// Optimizes request count per object.
// > If a single object has more than one request, these multiple requests can be handled via a single RPM-request.
METHOD PRIVATE OptimizeCOV : BOOL
VAR
	i : UDINT;
	j : UDINT;
	bSkipCov : BOOL;
END_VAR
IF (nReqList > 0) THEN
	FOR i:=0 TO nReqList-1 DO
		IF stReqList[i].iReq <> 0 AND_THEN F_IsCovReqType(stReqList[i].iReq) AND_THEN stReqList[i].fbCov^.Master = 0 THEN
			bSkipCov := F_IsCovProperty(stReqList[i].fbCov^.iObject.ObjectType, stReqList[i].fbCov^.ePropID);
			FOR j:=i+1 TO nReqList-1 DO
				IF stReqList[j].iReq <> 0 AND_THEN F_IsCovReqType(stReqList[j].iReq) AND_THEN stReqList[i].fbCov^.iObject.ObjectID = stReqList[j].fbCov^.iObject.ObjectID THEN
					 stReqList[i].fbCov^.AddCovSlave(stReqList[j].fbCov);
					 stReqList[j].fbCov^.Master:=stReqList[i].fbCov;
					 IF stReqList[j].fbCov^.fCOVIncrement = 0 AND F_IsCovProperty(stReqList[j].fbCov^.iObject.ObjectType, stReqList[j].fbCov^.ePropID) THEN
						 IF bSkipCov THEN
						 	stReqList[j].fbCov^.SendSubscription:=FALSE;
						 ELSE
							 bSkipCov:=TRUE;
						 END_IF
					 END_IF
				END_IF
			END_FOR
		END_IF
	END_FOR
END_IF
END_METHOD

// Called after online change.
{attribute 'call_after_online_change_slot' := '10'}
METHOD PROTECTED OnPostOnlineChange
IF iServer <> 0 THEN
	FW_SafeRelease(ADR(iServer));
	iServer:=0;
END_IF
IF iClient <> 0 THEN
	FW_SafeRelease(ADR(iClient));
	iClient:=0;
END_IF
iDevice:=0;

State:=E_BACnetRM_ClientState.eReInit;
END_METHOD

METHOD FB_Exit : BOOL
VAR_INPUT
	 bInCopyCode : BOOL; // if TRUE, the exit method is called for exiting an instance that is copied afterwards (online change).
END_VAR
IF iServer <> 0 THEN
	iServer.OnPlcAction(E_BACnet_PlcAction.eSuspend);
	iServer:=0;
END_IF
IF iClient <> 0 THEN
	FW_SafeRelease(ADR(iClient));
	iClient:=0;
END_IF

iDevice:=0;

DeleteReqList();

IF stReadList <> 0 THEN
	__DELETE(stReadList);
	stReadList:=0;
END_IF
IF stWriteList <> 0 THEN
	__DELETE(stWriteList);
	stWriteList:=0;
END_IF
END_METHOD

PROPERTY Error : BOOL
GET
Error := (eErrorID <> E_BACnet_Error.eNoError);
END_GET
END_PROPERTY

PROPERTY ObjectID : T_BACnet_ObjectIdentifier
GET
ObjectID := tObjectID;
END_GET
END_PROPERTY

PROPERTY ObjectInstance : UDINT
GET
ObjectInstance := nDeviceInstance;
END_GET
END_PROPERTY

PROPERTY ObjectType : E_BACnetObjType
GET
ObjectType := E_BACnetObjType.ObjDevice;
END_GET
END_PROPERTY

PROPERTY OpenRequestCount : UDINT
GET
OpenRequestCount:=nOpenReq;
END_GET
SET
nOpenReq:=OpenRequestCount;
END_SET
END_PROPERTY

PROPERTY ReadMode : E_BACnet_CommMode
GET
ReadMode:=eReadMode;
END_GET
SET
eReadMode:=ReadMode;
END_SET
END_PROPERTY

PROPERTY Ready : BOOL
GET
Ready := bReady;
END_GET
END_PROPERTY

PROPERTY State : E_BACnetRM_ClientState
GET
State := eState;
END_GET
SET
PRIVATE 
VAR
END_VAR
IF (State = E_BACnetRM_ClientState.eError) THEN
	_tReInitTime := TIME();
END_IF

eState := State;
END_SET
END_PROPERTY

END_FUNCTION_BLOCK

// POUs/Remote/Requests/[Internal]/FB_BACnetRM_ReqFifo
{attribute 'c++_compatible'}
{attribute 'enable_dynamic_creation'}
{attribute 'hide'}
FUNCTION_BLOCK FB_BACnetRM_ReqFifo EXTENDS FB_BACnetRM_ReqBase
VAR_INPUT
	bRpm : BOOL;
	bWpm : BOOL;
END_VAR
VAR
	pReqFifo	: POINTER TO ST_BACnetRM_FifoEntry;
	nReqFifo	: UDINT := 0;
	nMaxFifo	: UDINT := 0;
	nPendFifo	: UDINT := 0;
END_VAR

METHOD INTERNAL AddFifoReq : BOOL
VAR_INPUT
	pEntry : ST_BACnetRM_FifoEntry;
END_VAR
VAR
	nTmp : UDINT;
	nTmpSize : UDINT;
	pTmp : POINTER TO ST_BACnetRM_FifoEntry;
END_VAR
IF nReqFifo+1 >= nMaxFifo THEN
	nTmp := 2*nMaxFifo+100;
	nTmpSize := nTmp*SIZEOF(ST_BACnetRM_FifoEntry);
	pTmp := __NEW(BYTE,nTmpSize);
	IF pTmp = 0 THEN
		RETURN;
	END_IF
	IF pReqFifo <> 0 THEN
		MEMCPY(pTmp, pReqFifo, nMaxFifo*SIZEOF(ST_BACnetRM_FifoEntry));
		__DELETE(pReqFifo);
	END_IF
	pReqFifo:=pTmp;
	nMaxFifo:=nTmp;
END_IF

pReqFifo[nReqFifo]:=pEntry;
nReqFifo:=nReqFifo+1;

AddFifoReq:=TRUE;
END_METHOD

METHOD INTERNAL ProcessReadFifo : BOOL
VAR_INPUT
END_VAR
VAR
	pRequest : ST_BACnetRM_ReqPtr;
	nSize : UDINT;
	n :UDINT;
	pEntries : POINTER TO ST_BACnetRM_ReadEntry;	
	x : UDINT;
	iTmpFB : I_BACnetRM_BasicReq;
END_VAR
IF Valid THEN
	WHILE Client.nOpenReq < Client.nMaxParallelRequests AND nReqFifo > 0 DO		
		IF bRpm AND nReqFifo>1 THEN
			n:=0;
			nSize:=MIN(nReqFifo, Client.nRPMPropertiesPerRequest)*SIZEOF(ST_BACnetRM_ReadEntry);
			pRequest.fbRpm := __NEW(FB_BACnetRM_ReqRpm);
			IF pRequest.fbRpm = 0 THEN
				RETURN;
			END_IF
			pEntries:=__NEW(BYTE,nSize);
			IF pEntries = 0 THEN
				__DELETE(pRequest.fbRpm);
				RETURN;
			END_IF
			WHILE n<nReqFifo AND n < Client.nRPMPropertiesPerRequest DO
				pEntries[n].iObject:=pReqFifo[n].fbRead^.iObject;
				pEntries[n].ePropID:=pReqFifo[n].fbRead^.ePropID;
				pEntries[n].pData:=pReqFifo[n].fbRead^.pData;
				pEntries[n].nData:=pReqFifo[n].fbRead^.nData;
				pEntries[n].nIndex:=pReqFifo[n].fbRead^.nIndex;
				IF __QUERYINTERFACE(pReqFifo[0].fbRead^, iTmpFB) THEN
					pEntries[n].iReadFB:=iTmpFB;
				END_IF
				n:=n+1;
			END_WHILE		
			pRequest.fbRpm^(Client:=Client, iObject:=pReqFifo[0].fbRead^.iObject, pEntries:=pEntries, nEntries:=n, bFreeEntries:=TRUE);
			IF pRequest.fbRpm^.UpdateRequest() AND_THEN pRequest.fbRpm^.Send() THEN
				Client.OpenRequestCount:=Client.nOpenReq+1;
				pReqFifo[0].fbRead^.Request:=pRequest;
				pReqFifo[0].fbRead^.bRequestRPM:=TRUE;
				IF nReqFifo-n > 0 THEN
					MEMMOVE(pReqFifo, ADR(pReqFifo[n]), (nReqFifo-n)*SIZEOF(ST_BACnetRM_ReadEntry));
				END_IF
				nReqFifo:=nReqFifo-n;
			ELSE
				__DELETE(pRequest.fbRpm);
				RETURN;
			END_IF
		ELSE
			pRequest.fbRead := __NEW(FB_BACnetRM_ReqRead);
			IF pRequest.fbRead = 0 THEN
				RETURN;
			END_IF
			__QUERYINTERFACE(pReqFifo[0].fbRead^, iTmpFB);
			pRequest.fbRead^(Client:=Client, iObject:=pReqFifo[0].fbRead^.iObject, pData:=pReqFifo[0].fbRead^.pData, nData:=pReqFifo[0].fbRead^.nData, ePropID:=pReqFifo[0].fbRead^.ePropID, iReadFB:=iTmpFB);
			Client.OpenRequestCount:=Client.nOpenReq+1;
			pReqFifo[0].fbRead^.Request:=pRequest;	
			pReqFifo[0].fbRead^.bRequestRPM:=FALSE;
			IF pRequest.fbRead^.Send() THEN
				IF nReqFifo-n > 0 THEN
					MEMMOVE(pReqFifo, ADR(pReqFifo[1]),(nReqFifo-1)*SIZEOF(ST_BACnetRM_ReadEntry));
				END_IF
				nReqFifo:=nReqFifo-1;
			ELSE
				Client.OpenRequestCount:=Client.nOpenReq-1;
				__DELETE(pRequest.fbRead);
				RETURN;
			END_IF
		END_IF
	END_WHILE
	
	ProcessReadFifo:=TRUE;
ELSE
	// (BETA) ... Output Error
END_IF
END_METHOD

METHOD INTERNAL ProcessWriteFifo : BOOL
VAR_INPUT
END_VAR
VAR
	pRequest : ST_BACnetRM_ReqPtr;
	nSize : UDINT;
	n : UDINT;
	pEntries : POINTER TO ST_BACnetRM_WriteEntry;
	iTmpFB : I_BACnetRM_BasicReq;
END_VAR
IF Valid THEN
	WHILE Client.nOpenReq < Client.nMaxParallelRequests AND nReqFifo > 0 DO		
		IF bWpm THEN
			n:=0;
			nSize:=MIN(nReqFifo, Client.nRPMPropertiesPerRequest)*SIZEOF(ST_BACnetRM_WriteEntry);
			pRequest.fbWpm:= __NEW(FB_BACnetRM_ReqWpm);
			IF pRequest.fbWpm = 0 THEN
				RETURN;
			END_IF
			pEntries:=__NEW(BYTE,nSize);
			IF pEntries = 0 THEN
				__DELETE(pRequest.fbWpm);
				RETURN;
			END_IF
			WHILE n<nReqFifo-1 AND n < Client.nRPMPropertiesPerRequest DO
				pEntries[n].iObject:=pReqFifo[n].fbWrite^.iObject;
				pEntries[n].ePropID:=pReqFifo[n].fbWrite^.ePropID;
				pEntries[n].pData:=pReqFifo[n].fbWrite^.pData;
				pEntries[n].nData:=pReqFifo[n].fbWrite^.nData;
				pEntries[n].nIndex:=pReqFifo[n].fbWrite^.nIndex;
				IF __QUERYINTERFACE(pReqFifo[0].fbWrite^, iTmpFB) THEN
					pEntries[n].iWriteFB:=iTmpFB;
				END_IF
				n:=n+1;
			END_WHILE
			pRequest.fbWpm^(Client:=Client, pEntries:=pEntries, nEntries:=n, bFreeEntries:=TRUE);
			IF pRequest.fbWpm^.UpdateRequest() AND_THEN pRequest.fbWpm^.Send() THEN
				Client.OpenRequestCount:=Client.nOpenReq+1;
				pReqFifo[0].fbRead^.Request:=pRequest;
				pReqFifo[0].fbWrite^.bRequestWPM:=TRUE;
				IF nReqFifo-n > 0 THEN
					MEMMOVE(pReqFifo, ADR(pReqFifo[n]), (nReqFifo-n)*SIZEOF(ST_BACnetRM_WriteEntry));
				END_IF
				nReqFifo:=nReqFifo-n;
			ELSE
				__DELETE(pRequest.fbWpm);
				RETURN;
			END_IF
		ELSE
			pRequest.fbWrite := __NEW(FB_BACnetRM_ReqWrite);
			IF pRequest.fbWrite = 0 THEN
				RETURN;
			END_IF
			pRequest.fbWrite^.pData:=pReqFifo[0].fbWrite^.pData;
			pRequest.fbWrite^.nData:=pReqFifo[0].fbWrite^.nData;
			__QUERYINTERFACE(pReqFifo[0].fbWrite^, iTmpFB);
			pRequest.fbWrite^(Client:=Client, iObject:=pReqFifo[0].fbWrite^.iObject, ePropID:=pReqFifo[0].fbWrite^.ePropID, iWriteFB:=iTmpFB);
			IF pRequest.fbWrite^.Send() THEN
				pReqFifo[0].fbWrite^.Request:=pRequest;	
				pReqFifo[0].fbWrite^.bRequestWPM:=FALSE;
				Client.OpenRequestCount:=Client.nOpenReq+1;
				IF (nReqFifo-1) > 0 THEN
					MEMMOVE(pReqFifo, ADR(pReqFifo[1]),(nReqFifo-1)*SIZEOF(ST_BACnetRM_WriteEntry));
				END_IF
				nReqFifo:=nReqFifo-1;
			ELSE
				__DELETE(pRequest.fbWrite);
				RETURN;
			END_IF
		END_IF
	END_WHILE
	
	ProcessWriteFifo:=TRUE;
ELSE
	// (BETA) ... Output Error
END_IF
END_METHOD

METHOD FB_Exit : BOOL
VAR_INPUT
	 bInCopyCode : BOOL; // if TRUE, the exit method is called for exiting an instance that is copied afterwards (online change).
END_VAR
IF pReqFifo <> 0 THEN
	__DELETE(pReqFifo);
	pReqFifo:=0;
END_IF
END_METHOD

PROPERTY Valid : BOOL
GET
// Hint:
// > Don't call "super()"!
//   The "iObject" Interface-pointer is ignored to this instance because it is unused.
Valid := (__ISVALIDREF(Client));
END_GET
END_PROPERTY

END_FUNCTION_BLOCK

// POUs/Remote/Requests/[Internal]/[Base]/FB_BACnetRM_ReqBase
{attribute 'c++_compatible'}
{attribute 'enable_dynamic_creation'}
{attribute 'hide'}
FUNCTION_BLOCK FB_BACnetRM_ReqBase IMPLEMENTS I_BACnetRM_BaseReq
VAR_INPUT
	{attribute 'initialize_on_call'}
	{attribute 'no_copy'}
	Client : REFERENCE TO FB_BACnet_Client;
	iObject : I_BACnetRM_BaseObject;
END_VAR

METHOD PROTECTED OnError
VAR_INPUT
	stResult		: POINTER TO SendDataRequestResult;
	sLogCode		: STRING			:= '';
END_VAR
VAR
	i : UDINT;
END_VAR
IF (iObject <> 0) THEN
	iObject.OnReqError(THIS^, stResult, 'OE01');
END_IF
END_METHOD

METHOD GetRequestType : E_BACnetRM_RequestType
VAR_INPUT
END_VAR
GetRequestType:=E_BACnetRM_RequestType.eUndefined;
END_METHOD

METHOD IsReady : BOOL
END_METHOD

PROPERTY Valid : BOOL
GET
VAR
	iTest : BOOL;
END_VAR
Valid := (__ISVALIDREF(Client)) AND (iObject <> 0);
END_GET
END_PROPERTY

METHOD Send : BOOL
VAR
	_ClTmp : ITcIoBACnetPlcClient;
END_VAR
END_METHOD

END_FUNCTION_BLOCK

// POUs/Remote/Requests/[Internal]/FB_BACnetRM_ReqRpm
{attribute 'c++_compatible'}
{attribute 'enable_dynamic_creation'}
{attribute 'hide'}
FUNCTION_BLOCK FB_BACnetRM_ReqRpm EXTENDS FB_BACnetRM_ReqBasic
VAR_INPUT
	pEntries : POINTER TO ST_BACnetRM_ReadEntry;
	nEntries : UDINT;
	bFreeEntries : BOOL; 
END_VAR
VAR_OUTPUT
	bInit : BOOL;
END_VAR
VAR 
	req : SendDataRequest;
	pTmp : POINTER TO ST_BACnetRM_RpmListEntry;
END_VAR

IF NOT __ISVALIDREF(Client) THEN
	bError:=TRUE;
END_IF

SUPER^();

{attribute 'hide'}
METHOD Send : BOOL
IF Valid THEN
	IF stReq = 0 THEN
		RETURN;
	END_IF
	
	Send:=SUPER^.Send();
END_IF
END_METHOD

METHOD INTERNAL UpdateRequest : BOOL
VAR_INPUT
END_VAR
VAR
	nSize : UDINT;
	i : UDINT;
	nTmpSize : UDINT;
END_VAR
IF Valid THEN
	IF stReq <> 0 AND_THEN stReq^.pData <> 0 THEN
		pTmp:=stReq^.pData;
		__DELETE(pTmp);
		stReq^.pData:=0;
	END_IF
	nTmpSize := SIZEOF(ST_BACnetRM_RpmListEntry)*nEntries;
	pTmp := __NEW(BYTE,nTmpSize);
	IF pTmp = 0 THEN
		RETURN;
	END_IF
	
	FOR i:=0 TO nEntries-1 DO
		pTmp[i].tObjectID := pEntries[i].iObject.ObjectID;
		pTmp[i].ePropID := pEntries[i].ePropID;
		pTmp[i].nArrayIndex := 0;
		pTmp[i].nValidBits := 0;
		pTmp[i].nPriority := 0;
		pTmp[i].nEntrySize := SIZEOF(ST_BACnetRM_RpmListEntry) - 8;
		IF i <> nEntries -1 THEN
			pTmp[i].nEntrySize := pTmp[i].nEntrySize + 16#80000000;
		END_IF
	END_FOR
	
	stReq := ADR(req);
	stReq^.pData := pTmp;
	stReq^.nData := nTmpSize;
	
	stReq^.service := E_BACnetConfirmedService.SrvReadPropertyMultiple;
	stReq^.deviceId := Client.ObjectInstance;
	
	bInit:=TRUE;
	
	UpdateRequest:=TRUE;
ELSE
	// (BETA) ... Output Error
END_IF
END_METHOD

METHOD PRIVATE Free
VAR_INPUT
END_VAR
IF bFreeEntries AND pEntries <> 0 THEN
	__DELETE(pEntries);
	pEntries:=0;
	bFreeEntries:=FALSE;
END_IF

IF stReq <> 0 AND_THEN stReq^.pData <> 0 THEN
	pTmp:=req.pData;
	__DELETE(pTmp);
	req.pData:=0;
	stReq:=0;
END_IF
END_METHOD

METHOD PROTECTED OnError
VAR_INPUT
	stResult		: POINTER TO SendDataRequestResult;
	sLogCode		: STRING			:= '';
END_VAR
VAR
	i : UDINT;
END_VAR
// Do not call super! Handle each entry's error:
// SUPER^.OnError(eResult, sLogCode);

FOR i:=0 TO nEntries-1 DO
	IF pEntries[i].iReadFB <> 0 THEN
		pEntries[i].iReadFB.SetError();
		IF (pEntries[i].iObject <> 0) THEN
			pEntries[i].iObject.OnReqError(THIS^, stResult, 'OE07');
		END_IF	
	END_IF
END_FOR
END_METHOD

METHOD PROTECTED ProcessResult : HRESULT
VAR_INPUT
	pResult	: POINTER TO SendDataRequestResult;
END_VAR
VAR
	pPropList : POINTER TO ST_BACnetRM_RpmListEntry;
	i : UDINT;
END_VAR
IF pResult^.service <> E_BACnetConfirmedService.SrvReadPropertyMultiple THEN
	ProcessResult:=E_FAIL;
	RETURN;
END_IF

IF pEntries = 0 THEN // Request object has already been deleted
	ProcessResult:=E_FAIL;
	RETURN;
END_IF

// set all entries to error, all good entries in response will be set to good afterwards
FOR i:=0 TO nEntries-1 DO
	IF pEntries[i].iReadFB <> 0 THEN
		pEntries[i].iReadFB.SetError();
	END_IF
	
	pEntries[i]._bError := TRUE;
END_FOR

// copy data:
pPropList := pResult^.pData;
WHILE pPropList <> 0 DO
	_WritePropEntry(pPropList);
	pPropList := F_BACnet_NextListElem(pPropList, pPropList^.nEntrySize);
END_WHILE

// Evaluate remaining errors:
FOR i:=0 TO nEntries-1 DO
	IF (pEntries[i]._bError) AND_THEN (pEntries[i].iObject <> 0) THEN
		pEntries[i].iObject.OnReqError(THIS^, pResult, 'OE28');
	END_IF
END_FOR

ProcessResult:=S_OK;
END_METHOD

METHOD PRIVATE _WritePropEntry : BOOL
VAR_INPUT
	pEntry : POINTER TO ST_BACnetRM_RpmListEntry;
END_VAR
VAR
	i : UDINT;
END_VAR
FOR i:=0 TO nEntries-1 DO
	IF (pEntries[i].iObject.ObjectID = pEntry^.tObjectID) AND (pEntries[i].ePropID = pEntry^.ePropID) THEN
		CopyRemoteData(pEntries[i].iObject, pEntry^.ePropID ,pEntries[i].pData, pEntries[i].nData, F_BACnet_EndOf(pEntry, SIZEOF(ST_BACnetRM_RpmListEntry)), F_BACnet_ElemSize(pEntry^.nEntrySize)-16); 
		IF pEntries[i].iReadFB <> 0 THEN
			pEntries[i].iReadFB.SetReady();
		END_IF
		pEntries[i]._bError := FALSE;
		
		_WritePropEntry:=TRUE;
	END_IF
END_FOR
END_METHOD

METHOD FB_exit : BOOL
VAR_INPUT
	bInCopyCode : BOOL; // if TRUE, the exit method is called for exiting an instance that is copied afterwards (online change).
END_VAR
Free();
END_METHOD

METHOD GetRequestType : E_BACnetRM_RequestType
VAR_INPUT
END_VAR
GetRequestType := E_BACnetRM_RequestType.eReadPropertyMultiple;
END_METHOD

END_FUNCTION_BLOCK

// POUs/Remote/Requests/[Internal]/[Base]/FB_BACnetRM_ReqBasic
{attribute 'c++_compatible'}
{attribute 'enable_dynamic_creation'}
{attribute 'hide'}
FUNCTION_BLOCK FB_BACnetRM_ReqBasic EXTENDS FB_BACnetRM_ReqBase IMPLEMENTS ITcIoBACnetServiceResponseSink
VAR_INPUT
	tCycleTime : TIME := T#5S;
END_VAR
VAR_OUTPUT
	bBusy : BOOL;
	bError : BOOL;
	bReady : BOOL;
END_VAR
VAR
	{attribute 'hide'}
	stReq : POINTER TO SendDataRequest;
	timer : TON;
END_VAR

{attribute 'c++_compatible'}
{attribute 'minimal_input_size' := '4'}
{attribute 'pack_mode' := '4'}
{attribute 'hide'}
METHOD OnSendPropertyDataRequest : HRESULT
VAR_INPUT
	pResult	: POINTER TO SendDataRequestResult;
END_VAR
IF (Valid) AND_THEN (pResult <> 0) THEN
	IF F_BACnetRM_IsErrorSet(pResult) THEN
		SetError();
		OnError(pResult, 'OSPDR04');
		OnSendPropertyDataRequest:=S_FALSE;
	ELSE
		IF S_OK = ProcessResult(pResult) THEN
			SetReady();
			OnSendPropertyDataRequest:=S_OK;
		ELSE
			OnSendPropertyDataRequest:=S_FALSE;
		END_IF	
	END_IF
	Client.OnRequestComplete();
END_IF
END_METHOD

METHOD INTERNAL InitTimer : BOOL
VAR_INPUT
END_VAR
timer(IN:=FALSE, PT:=T#1MS);
timer(IN:=TRUE, PT:=T#1MS);
END_METHOD

{attribute 'hide'}
METHOD SetBusy
bBusy := TRUE;
bError := FALSE;
bReady := FALSE;
END_METHOD

{attribute 'hide'}
METHOD SetError
bBusy := FALSE;
bError := TRUE;
bReady := FALSE;
END_METHOD

{attribute 'hide'}
METHOD SetReady
bBusy := FALSE;
bError := FALSE;
bReady := TRUE;
END_METHOD

{attribute 'c++_compatible'}
{attribute 'minimal_input_size' := '4'}
{attribute 'pack_mode' := '4'}
{attribute 'hide'}
METHOD TcAddRef : UDINT
END_METHOD

{attribute 'c++_compatible'}
{attribute 'minimal_input_size' := '4'}
{attribute 'pack_mode' := '4'}
{attribute 'hide'}
METHOD TcQueryInterface : HRESULT
VAR_INPUT
	iid	: REFERENCE TO IID;
	pipItf	: POINTER TO PVOID;
END_VAR
VAR
	ipSink : ITcIoBACnetServiceResponseSink;
	ipUnknown : ITcUnknown;	
END_VAR
IF GuidsEqual(ADR(iid), ADR(TC_GLOBAL_IID_LIST.IID_ITcIoBACnetServiceResponseSink)) THEN
	ipSink := THIS^; // cast to interface pointer
	pipItf^ := ITCUNKNOWN_TO_PVOID(ipSink);
	TcAddRef();
	TcQueryInterface := S_OK;
ELSIF GuidsEqual(ADR(iid), ADR(TC_GLOBAL_IID_LIST.IID_ITcUnknown)) THEN
	ipUnknown := THIS^; // cast to interface pointer
	pipItf^ := ITCUNKNOWN_TO_PVOID(ipUnknown);
	TcAddRef();
	TcQueryInterface := S_OK;
ELSE
	TcQueryInterface := E_HRESULTAdsErr.NOINTERFACE ; //Call super if this fb extends some other
END_IF
END_METHOD

{attribute 'c++_compatible'}
{attribute 'minimal_input_size' := '4'}
{attribute 'pack_mode' := '4'}
{attribute 'hide'}
METHOD TcRelease : UDINT
END_METHOD

METHOD PROTECTED CopyRemoteData : BOOL
VAR_INPUT
	iObject : I_BACnetRM_BaseObject;
	ePropID : E_BACnetPropIdentifier;
	pDst : PVOID;
	nDst : UDINT;
	pRead : PVOID;
	nRead : UDINT;
END_VAR
VAR
	i 	 : INT;
	pByte : POINTER TO BYTE;
	pSchedPv : POINTER TO ST_BACnet_ValueList;
END_VAR
// Individual treatment:
CASE (ePropID) OF
	E_BACnetPropIdentifier.PropPresentValue:
		IF iObject.ObjectType = E_BACnetObjType.ObjSchedule THEN
			IF (nRead >= 16) THEN
				pSchedPv := pRead;
				CASE pSchedPv^.listEntry.eValueChoice OF
					E_BACnet_ValueChoice.eBoolValue:
						MEMCPY(pDst, ADR(pSchedPv^.listEntry.stValue), MIN(SIZEOF(BOOL),nDst)); 
					E_BACnet_ValueChoice.eRealValue:
						MEMCPY(pDst, ADR(pSchedPv^.listEntry.stValue), MIN(SIZEOF(REAL),nDst)); 
					E_BACnet_ValueChoice.eUnsignedValue:
						MEMCPY(pDst, ADR(pSchedPv^.listEntry.stValue), MIN(SIZEOF(UDINT),nDst)); 
					E_BACnet_ValueChoice.eEnumerationValue:
						MEMCPY(pDst, ADR(pSchedPv^.listEntry.stValue.enumValue), MIN(SIZEOF(UDINT),nDst)); 
				END_CASE
			
				CopyRemoteData := TRUE;
			END_IF
		END_IF
		
	// Consider enumerations with smaller base-types:
	E_BACnetPropIdentifier.PropCurrentlyActivePriority:
		nRead := nDst;
		
END_CASE

// Check if received bytes match expected size:
IF (NOT CopyRemoteData) AND_THEN (nRead <= nDst) THEN
	// Individual treatment:
	CASE (ePropID) OF
		E_BACnetPropIdentifier.PropStatusFlags:
			pByte:=pDst;
			FOR i:=0 TO 3 DO
				IF F_BACnet_IsBitFieldBitSetPtr(pRead, i) THEN
					pByte[i]:=1;
				ELSE
					pByte[i]:=0;
				END_IF
			END_FOR
			
		E_BACnetPropIdentifier.PropAckedTransitions,
		E_BACnetPropIdentifier.PropEventEnable:
			pByte:=pDst;
			FOR i:=0 TO 2 DO
				IF F_BACnet_IsBitFieldBitSetPtr(pRead, i) THEN
					pByte[i]:=1;
				ELSE
					pByte[i]:=0;
				END_IF
			END_FOR
			
	ELSE
		// Default treatment:
		MEMCPY(pDst, pRead, MIN(nRead,nDst)); 
	END_CASE
	
	CopyRemoteData := TRUE;
END_IF

IF (CopyRemoteData) THEN
	// Notify object about changed value:
	iObject.OnCOV(ePropID);
ELSE
	F_BA_LogMessage3(ADSLOG_MSGTYPE_ERROR, 'CRD51', 'Unable to process remote data due to invalid size (Property: "%d", Read: %d Bytes, Expected: %d Bytes)!', F_INT(ePropID), F_UDINT(nRead), F_UDINT(nDst));
END_IF
END_METHOD

METHOD PROTECTED ProcessResult : HRESULT
VAR_INPUT
	pResult	: POINTER TO SendDataRequestResult;
END_VAR
ProcessResult:=S_OK;
END_METHOD

METHOD Send : BOOL
VAR
	_ClTmp : ITcIoBACnetPlcClient;
END_VAR
IF Valid THEN
	_ClTmp := Client.iClient;
	
	SetBusy();
	IF S_OK = _ClTmp.SendPropertyDataRequest(stReq, THIS^) THEN
		Send:=TRUE;
		StartTimer();
	ELSE
		SetError();
		Send:=FALSE; 
	END_IF
END_IF
END_METHOD

METHOD PROTECTED StartTimer : BOOL
VAR_INPUT
END_VAR
timer(IN:=FALSE, PT:=tCycleTime);
timer(IN:=TRUE, PT:=tCycleTime);
END_METHOD

METHOD GetRequestType : E_BACnetRM_RequestType
VAR_INPUT
END_VAR
GetRequestType:=E_BACnetRM_RequestType.eUndefined;
END_METHOD

METHOD IsReady : BOOL
VAR_INPUT
END_VAR
timer(Q=>IsReady);
IF bBusy THEN
	IsReady:=FALSE;
END_IF
END_METHOD

END_FUNCTION_BLOCK

// POUs/Remote/Requests/[Internal]/FB_BACnetRM_ReqRead
{attribute 'c++_compatible'}
{attribute 'enable_dynamic_creation'}
{attribute 'hide'}
FUNCTION_BLOCK FB_BACnetRM_ReqRead EXTENDS FB_BACnetRM_ReqBasic
VAR_INPUT
	ePropID : E_BACnetPropIdentifier;
	pData : PVOID;
	nData : UDINT;
	iReadFB : I_BACnetRM_BasicReq;
END_VAR
VAR 
	req : SendDataRequest;
END_VAR

IF NOT __ISVALIDREF(Client) THEN
	bError:=TRUE;
END_IF

SUPER^();

{attribute 'hide'}
METHOD Send : BOOL
IF Valid THEN
	IF stReq = 0 THEN
		IF ePropID = E_BACnetPropIdentifier.PropLogBuffer THEN
			req.service := E_BACnetConfirmedService.SrvReadRange;
		ELSE
			req.service := E_BACnetConfirmedService.SrvReadProperty;
		END_IF	
		req.objectIdentifier := iObject.ObjectID;
		req.propertyIdentifier := ePropID;
		req.pData := pData;
		req.nData := nData;
		req.deviceId := Client.ObjectInstance;
		stReq := ADR(req);
	END_IF
	
	Send:=SUPER^.Send();
END_IF
END_METHOD

METHOD PROTECTED OnError
VAR_INPUT
	stResult		: POINTER TO SendDataRequestResult;
	sLogCode		: STRING			:= '';
END_VAR
SUPER^.OnError(stResult, sLogCode);

IF iReadFB <> 0 THEN
	iReadFB.SetError();
END_IF
END_METHOD

METHOD PROTECTED ProcessResult : HRESULT
VAR_INPUT
	pResult	: POINTER TO SendDataRequestResult;
END_VAR
IF Valid THEN
	IF (CopyRemoteData(iObject, ePropID, pData, nData, pResult^.pData, pResult^.nData)) THEN
		IF iReadFB <> 0 THEN
			iReadFB.SetReady();
		END_IF
		ProcessResult:=S_OK;
	ELSE
		IF iReadFB <> 0 THEN
			iReadFB.SetError();
		END_IF
		ProcessResult:=E_FAIL;
	END_IF
END_IF
END_METHOD

METHOD GetRequestType : E_BACnetRM_RequestType
VAR_INPUT
END_VAR
GetRequestType:=E_BACnetRM_RequestType.eRead;
END_METHOD

END_FUNCTION_BLOCK

// POUs/Remote/Requests/[Internal]/FB_BACnetRM_ReqWpm
{attribute 'c++_compatible'}
{attribute 'enable_dynamic_creation'}
{attribute 'hide'}
FUNCTION_BLOCK FB_BACnetRM_ReqWpm EXTENDS FB_BACnetRM_ReqBasic
VAR_INPUT
	pEntries : POINTER TO ST_BACnetRM_WriteEntry;
	nEntries : UDINT;
	bFreeEntries : BOOL; 
END_VAR
VAR_OUTPUT
	bInit : BOOL;
END_VAR
VAR 
	{attribute 'hide'}
	req : SendDataRequest;
	{attribute 'hide'}
	pTmp : POINTER TO ST_BACnetRM_RpmListEntry;
END_VAR

IF NOT __ISVALIDREF(Client) THEN
	bError:=TRUE;
END_IF

SUPER^();

{attribute 'hide'}
METHOD Send : BOOL
IF Valid THEN
	IF stReq = 0 THEN
		Send:=FALSE;
		RETURN;
	END_IF
	
	UpdateRequest();
	Send:=SUPER^.Send();
END_IF
END_METHOD

METHOD INTERNAL UpdateRequest : BOOL
VAR_INPUT
END_VAR
VAR
	nSize : UDINT;
	i : UDINT;
	nTmpSize : UDINT;
	nTmpEntrySize : UDINT;
END_VAR
IF Valid THEN
	IF stReq <> 0 AND_THEN stReq^.pData <> 0 THEN
		pTmp:=stReq^.pData;
		__DELETE(pTmp);
	END_IF
	FOR i:=0 TO nEntries-1 DO
		IF pEntries[i].pEnable = 0 OR_ELSE pEntries[i].pEnable^ > 0 THEN
			nTmpSize := nTmpSize + SIZEOF(ST_BACnetRM_RpmListEntry) + F_BACnet_AlignedSize(F_BACnetRM_GetWriteEntrySize(pEntries[i]));
		END_IF
	END_FOR
	pTmp := __NEW(BYTE,nTmpSize);
	IF pTmp = 0 THEN
		UpdateRequest:=FALSE;
		RETURN;
	END_IF
	
	stReq := ADR(req);
	stReq^.pData := pTmp;
	FOR i:=0 TO nEntries-1 DO
		IF pEntries[i].pEnable = 0 OR_ELSE pEntries[i].pEnable^ > 0 THEN
			pTmp^.tObjectID := pEntries[i].iObject.ObjectID;
			pTmp^.ePropID := pEntries[i].ePropID;
			pTmp^.nArrayIndex := 0;
			pTmp^.nValidBits := 0; 
			IF pEntries[i].nPriority <> 16 THEN
				pTmp^.nValidBits.1 := 1;
				pTmp^.nPriority := pEntries[i].nPriority;
			ELSE
				pTmp^.nPriority := 0;
			END_IF
			nTmpEntrySize := F_BACnetRM_GetWriteEntrySize(pEntries[i]);
			pTmp^.nEntrySize := F_BACnet_AlignedSize(nTmpEntrySize) + SIZEOF(ST_BACnetRM_RpmListEntry) - 8;
			
			IF nTmpEntrySize <> 0 THEN
				MEMCPY(F_BACnet_EndOf(pTmp, SIZEOF(ST_BACnetRM_RpmListEntry)), pEntries[i].pData, pEntries[i].nData); 
			END_IF

			IF i <> nEntries -1 THEN
				pTmp[i].nEntrySize := pTmp[i].nEntrySize + 16#80000000;
			END_IF
			pTmp := F_BACnet_NextListElem(pTmp, pTmp^.nEntrySize);
		END_IF
	END_FOR
	
	stReq^.nData := nTmpSize;
	stReq^.service := E_BACnetConfirmedService.SrvWritePropertyMultiple;
	stReq^.deviceId := Client.ObjectInstance;
	
	bInit:=TRUE;
	
	UpdateRequest:=TRUE;
ELSE
	F_BA_LogMessage(ADSLOG_MSGTYPE_ERROR, 'WPM82', 'WPM Request not valid!');
END_IF
END_METHOD

METHOD PRIVATE Free
VAR_INPUT
END_VAR
IF bFreeEntries AND pEntries <> 0 THEN
	__DELETE(pEntries);
	pEntries:=0;
	bFreeEntries:=FALSE;
END_IF

IF stReq <> 0 AND_THEN stReq^.pData <> 0 THEN
	pTmp:=req.pData;
	__DELETE(pTmp);
	req.pData:=0;
	stReq:=0;
END_IF
END_METHOD

METHOD PROTECTED OnError
VAR_INPUT
	stResult		: POINTER TO SendDataRequestResult;
	sLogCode		: STRING			:= '';
END_VAR
VAR
	i : UDINT;
END_VAR
// Do not call super! Handle each entry's error:
// SUPER^.OnError(eResult, sLogCode);

FOR i:=0 TO nEntries-1 DO
	IF pEntries[i].iWriteFB <> 0 THEN
		pEntries[i].iWriteFB.SetError();
		IF (pEntries[i].iObject <> 0) THEN
			pEntries[i].iObject.OnReqError(THIS^, stResult, 'OE10');
		END_IF		
	END_IF
END_FOR
END_METHOD

METHOD PROTECTED ProcessResult : HRESULT
VAR_INPUT
	pResult	: POINTER TO SendDataRequestResult;
END_VAR
VAR
	pPropList : POINTER TO ST_BACnetRM_RpmListEntry;
END_VAR
VAR
	i : UDINT;
END_VAR
IF pResult^.service <> E_BACnetConfirmedService.SrvWritePropertyMultiple THEN
	SetError();
	RETURN;
END_IF

FOR i:=0 TO nEntries-1 DO
	IF pEntries[i].iWriteFB <> 0 THEN
		pEntries[i].iWriteFB.SetReady();	// TODO: handle error entry		
	END_IF
END_FOR
SetReady();
END_METHOD

METHOD FB_exit : BOOL
VAR_INPUT
	bInCopyCode : BOOL; // if TRUE, the exit method is called for exiting an instance that is copied afterwards (online change).
END_VAR
Free();
END_METHOD

METHOD GetRequestType : E_BACnetRM_RequestType
VAR_INPUT
END_VAR
GetRequestType := E_BACnetRM_RequestType.eWritePropertyMultiple;
END_METHOD

END_FUNCTION_BLOCK

// POUs/Remote/Requests/[Internal]/FB_BACnetRM_ReqWrite
{attribute 'c++_compatible'}
{attribute 'enable_dynamic_creation'}
{attribute 'hide'}
FUNCTION_BLOCK FB_BACnetRM_ReqWrite EXTENDS FB_BACnetRM_ReqBasic
VAR_INPUT CONSTANT
	ePropID : E_BACnetPropIdentifier;
	pData : PVOID;
	nData : UDINT;
	pEnable : POINTER TO BOOL;
	pNull : POINTER TO BOOL;
	fCOVIncrement : REAL;
	ePriority : E_BACnet_Priority := E_BACnet_Priority.Last;
	{attribute 'hide'}
	iWriteFB : I_BACnetRM_BasicReq;
END_VAR
VAR 
	{attribute 'hide'}
	req : SendDataRequest;
	{attribute 'hide'}
	lastWriteValue : ST_BACnetRM_LastWriteValue;
	{attribute 'hide'}
	bInstData : UDINT;
END_VAR
VAR_STAT
	// (BETA) ... Following symbols should be made non-static / thread safe!
	{region 'Temporary'}
		{attribute 'hide'}
		_bEn : POINTER TO BOOL;
	{endregion}	
END_VAR

IF NOT __ISVALIDREF(Client) THEN
	bError:=TRUE;
END_IF

SUPER^();

{attribute 'hide'}
METHOD Send : BOOL
VAR
END_VAR
IF Valid THEN
	IF (pData <> 0) THEN
		IF stReq = 0 THEN
			req.service := E_BACnetConfirmedService.SrvWriteProperty;
			req.objectIdentifier := iObject.ObjectID;
			req.propertyIdentifier := ePropID;
			IF (F_BACnet_IsPriorityValid(ePriority)) THEN
				req.priority := TO_UDINT(ePriority);
			END_IF
			req.pData := pData;
			req.nData := nData;
			req.deviceId := Client.ObjectInstance;
			stReq := ADR(req);
		END_IF
		
		IF pNull <> 0 AND_THEN pNull^ THEN
			req.nData := 0;
		ELSE
			req.nData := nData;
		END_IF
		
		IF SUPER^.Send() THEN
			IF pNull <> 0 THEN
				lastWriteValue.stCmdValue.bNull := pNull^;
				IF nData <= 4 THEN
					MEMCPY(ADR(lastWriteValue.stCmdValue.fValue), pData, nData);
				ELSIF lastWriteValue.nOther <> 0 THEN
					MEMCPY(lastWriteValue.nOther, pData, nData);
				END_IF
			ELSE
				IF nData <= 4 THEN
					MEMCPY(ADR(lastWriteValue.n32Value), pData, nData);
				ELSIF lastWriteValue.nOther <> 0 THEN
					MEMCPY(lastWriteValue.nOther, pData, nData);
				END_IF
			END_IF
			Send:=TRUE;
		END_IF
	END_IF
END_IF
END_METHOD

METHOD PROTECTED OnError
VAR_INPUT
	stResult		: POINTER TO SendDataRequestResult;
	sLogCode		: STRING			:= '';
END_VAR
SUPER^.OnError(stResult, sLogCode);

IF iWriteFB <> 0 THEN
	iWriteFB.SetError();
END_IF
END_METHOD

METHOD PROTECTED ProcessResult : HRESULT
VAR_INPUT
	pResult	: POINTER TO SendDataRequestResult;
END_VAR
bReady:=TRUE;

IF iWriteFB <> 0 THEN
	iWriteFB.SetReady();
END_IF

ProcessResult:=S_OK;
END_METHOD

METHOD GetRequestType : E_BACnetRM_RequestType
VAR_INPUT
END_VAR
GetRequestType := E_BACnetRM_RequestType.eWrite;
END_METHOD

METHOD IsReady : BOOL
VAR_INPUT
END_VAR
VAR
	_fValue : REAL;
END_VAR
IF SUPER^.IsReady() THEN
	IF pEnable = 0 OR_ELSE pEnable^ THEN		
		IF fCOVIncrement <> 0.0 THEN
			MEMCPY(ADR(_fValue), pData, SIZEOF(_fValue));
			IF ABS(lastWriteValue.stCmdValue.fValue - _fValue) > fCOVIncrement THEN
				IF pNull = 0 OR_ELSE NOT pNull^ THEN
					IsReady:=TRUE;
					RETURN;
				END_IF
			END_IF
		ELSE
			IF MEMCMP(ADR(lastWriteValue.n32Value), pData, nData) <> 0 THEN 
				IF pNull = 0 OR_ELSE NOT pNull^ THEN
					IsReady:=TRUE;
					RETURN;
				END_IF
			END_IF
		END_IF
		IF pNull <> 0 AND_THEN pNull^ <> lastWriteValue.stCmdValue.bNull THEN
			IsReady:=TRUE;
			RETURN;
		END_IF
	END_IF
END_IF
END_METHOD

END_FUNCTION_BLOCK

// POUs/Remote/Properties/FB_BACnetRM_ReadProperty
FUNCTION_BLOCK FB_BACnetRM_ReadProperty EXTENDS FB_BACnetRM_BaseProperty
VAR_INPUT CONSTANT
	{attribute 'initialize_on_call'}
	{attribute 'no_copy'}
	Client : REFERENCE TO FB_BACnet_Client;
	bRequestRPM : BOOL;
END_VAR

SUPER^();

METHOD PROTECTED OnExecuteChange : BOOL
OnExecuteChange := Client.AddFifoReadReq(THIS);
END_METHOD

METHOD PROTECTED Free : BOOL
IF pRequest.pPtr <> 0 THEN
	IF bRequestRPM AND pRequest.fbRpm <> 0 THEN
		__DELETE(pRequest.fbRpm);
		pRequest.fbRpm:=0;
	ELSIF pRequest.fbRead <> 0 THEN
		__DELETE(pRequest.fbRead);
		pRequest.fbRead:=0;
	END_IF
	pRequest.pPtr:=0;
END_IF
END_METHOD

METHOD FB_exit : BOOL
VAR_INPUT
	bInCopyCode : BOOL; // if TRUE, the exit method is called for exiting an instance that is copied afterwards (online change).
END_VAR
Free();
END_METHOD

PROPERTY Valid : BOOL
GET
Valid := __ISVALIDREF(Client);
END_GET
END_PROPERTY

END_FUNCTION_BLOCK

// POUs/Remote/Properties/[Base]/FB_BACnetRM_BaseProperty
FUNCTION_BLOCK FB_BACnetRM_BaseProperty IMPLEMENTS I_BACnetRM_BasicReq
VAR_INPUT CONSTANT
	pData : PVOID;
	nData : UDINT;
	iObject : I_BACnetRM_BaseObject;
	nIndex : UDINT := 16#FFFFFFFF;
	ePropID : E_BACnetPropIdentifier;
	bExecute : BOOL;
	{attribute 'hide'}
	pRequest : ST_BACnetRM_ReqPtr;
END_VAR
VAR_OUTPUT
	bReady : BOOL;
	bBusy : BOOL;
	bError : BOOL;
END_VAR
VAR
	{attribute 'hide'}
	bExecuteOld : BOOL;
END_VAR

IF bExecuteOld <> bExecute THEN
	bExecuteOld := bExecute;

	IF NOT Valid THEN
		SetError();
	END_IF
	
	IF bExecute THEN
		IF bBusy THEN
			RETURN;
		END_IF
		Free();
		IF NOT OnExecuteChange() THEN
			SetError();
		ELSE
			SetBusy();
		END_IF
	ELSE
		bReady:=FALSE;
	END_IF
END_IF

{attribute 'hide'}
METHOD SetBusy
bBusy := TRUE;
bError := FALSE;
bReady := FALSE;
END_METHOD

{attribute 'hide'}
METHOD SetError
bBusy := FALSE;
bError := TRUE;
bReady := FALSE;
END_METHOD

{attribute 'hide'}
METHOD SetReady
bBusy := FALSE;
bError := FALSE;
bReady := TRUE;
END_METHOD

METHOD PROTECTED OnExecuteChange : BOOL
OnExecuteChange := FALSE;
END_METHOD

METHOD PROTECTED Free : BOOL
Free := FALSE;
END_METHOD

PROPERTY Busy : BOOL
GET
Busy:=bBusy;
END_GET
SET
bBusy:=Busy;
END_SET
END_PROPERTY

PROPERTY Error : BOOL
GET
Error:=bError;
END_GET
SET
bError:=Error;
END_SET
END_PROPERTY

PROPERTY Ready : BOOL
GET
Ready:=bReady;
END_GET
SET
bReady:=Ready;
END_SET
END_PROPERTY

PROPERTY Request : ST_BACnetRM_ReqPtr;
GET
Request:=pRequest;
END_GET
SET
pRequest:=Request;
END_SET
END_PROPERTY

PROPERTY Valid : BOOL
GET
Valid := FALSE;
END_GET
END_PROPERTY

END_FUNCTION_BLOCK

// POUs/Remote/Properties/FB_BACnetRM_WriteProperty
FUNCTION_BLOCK FB_BACnetRM_WriteProperty EXTENDS FB_BACnetRM_BaseProperty
VAR_INPUT CONSTANT
	{attribute 'initialize_on_call'}
	{attribute 'no_copy'}
	Client : REFERENCE TO FB_BACnet_Client;
	
	bRequestWPM : BOOL;
END_VAR

SUPER^();

METHOD PROTECTED OnExecuteChange : BOOL
OnExecuteChange := Client.AddFifoWriteReq(THIS);
END_METHOD

METHOD PROTECTED Free : BOOL
IF pRequest.pPtr <> 0 THEN
	IF bRequestWPM  AND pRequest.fbWpm <> 0 THEN
		__DELETE(pRequest.fbWpm);
		pRequest.fbWpm:=0;
	ELSIF pRequest.fbWrite <> 0 THEN
		__DELETE(pRequest.fbWrite);
		pRequest.fbWrite:=0;
	END_IF
	pRequest.pPtr:=0;
END_IF
END_METHOD

METHOD FB_exit : BOOL
VAR_INPUT
	bInCopyCode : BOOL; // if TRUE, the exit method is called for exiting an instance that is copied afterwards (online change).
END_VAR
Free();
END_METHOD

PROPERTY Valid : BOOL
GET
Valid := __ISVALIDREF(Client);
END_GET
END_PROPERTY

END_FUNCTION_BLOCK

// POUs/Remote/Requests/[Internal]/FB_BACnetRM_ReqCov
{attribute 'c++_compatible'}
{attribute 'enable_dynamic_creation'}
{attribute 'hide'}
{attribute 'hide'}
FUNCTION_BLOCK FB_BACnetRM_ReqCov EXTENDS FB_BACnetRM_ReqBasic
VAR_INPUT CONSTANT
	bConfirmed : BOOL;
	bUnsubscribed : BOOL;
	tLifetime : TIME := T#300S;
	fCOVIncrement : REAL := 0;
END_VAR
VAR_INPUT
	ePropID : E_BACnetPropIdentifier;
	pData : PVOID;
	nData : UDINT;
END_VAR
VAR_OUTPUT
	bSubsReady : BOOL;
END_VAR
VAR 
	req : SubscribeCovPropertyRequest;
	bSendSubs : BOOL := TRUE;
	pMaster : POINTER TO FB_BACnetRM_ReqCov;
	pCovSlaves : POINTER TO POINTER TO FB_BACnetRM_ReqCov;
	nCovSlaves : UDINT;
	nCovSlavesMax : UDINT;
END_VAR

IF NOT __ISVALIDREF(Client) THEN
	bError:=TRUE;
END_IF

SUPER^();

METHOD INTERNAL AddCovSlave : BOOL
VAR_INPUT
	pSlave : POINTER TO FB_BACnetRM_ReqCov;
END_VAR
VAR
	nTmp : UDINT;
	nTmpSize : UDINT;
	pTmp : POINTER TO POINTER TO FB_BACnetRM_ReqCov;
END_VAR
IF nCovSlaves+1 >= nCovSlavesMax THEN
	nTmp := nCovSlavesMax+10;
	nTmpSize := nTmp*SIZEOF(POINTER TO FB_BACnetRM_ReqCov);
	pTmp := __NEW(BYTE,nTmpSize);
	IF pTmp = 0 THEN
		RETURN;
	END_IF
	IF pCovSlaves <> 0 THEN
		MEMCPY(pTmp, pCovSlaves, nCovSlavesMax*SIZEOF(POINTER TO FB_BACnetRM_ReqCov));
		__DELETE(pCovSlaves);
	END_IF
	pCovSlaves:=pTmp;
	nCovSlavesMax:=nTmp;
END_IF

pCovSlaves[nCovSlaves]:=pSlave;
nCovSlaves:=nCovSlaves+1;
END_METHOD

{attribute 'hide'}
METHOD Send : BOOL
VAR
	iClientTmp : ITcIoBACnetPlcClient;
END_VAR
IF Valid THEN
	IF NOT bSendSubs THEN
		RETURN;
	END_IF
	
	IF stReq = 0 THEN
		IF bUnsubscribed THEN
			req.issueConfirmedNotifications := FALSE;
			req.lifetime := 0;
			req.subscriberProcessIdentifier := 0;
		ELSE
			req.issueConfirmedNotifications := bConfirmed;
			req.lifetime := TIME_TO_DWORD(tLifetime) / 500;
			req.subscriberProcessIdentifier := 1;
		END_IF
		req.monitoredObjectIdentifier := iObject.ObjectID;
		req.covIncrement := fCOVIncrement;
		req.monitoredPropertyIdentifier.propertyIdentifier := ePropID;
		req.monitoredPropertyIdentifier.validFields := 1;	
	
		req.validFields := 2#0011111;
		IF req.covIncrement <> 0 THEN
			req.validFields := req.validFields +  2#100000;
		END_IF
	END_IF
	
	iClientTmp := Client.iClient;
	IF S_OK = iClientTmp.SendCOVSubscription(ADR(req), THIS^) THEN
		Send:=TRUE;
		StartTimer();
	END_IF
END_IF
END_METHOD

METHOD PROTECTED ProcessResult : HRESULT
VAR_INPUT
	pResult	: POINTER TO SendDataRequestResult;
END_VAR
VAR
	pPropList : POINTER TO ST_BACnetRM_PropertyValueList;
	i : UDINT;
END_VAR
IF Valid THEN
	IF pResult^.service = E_BACnetConfirmedService.SrvSubscribeCOV OR pResult^.service = E_BACnetConfirmedService.SrvSubscribeCOVProperty THEN
		bSubsReady:=TRUE;
		RETURN;
	END_IF
	
	ProcessResult:=E_FAIL;
	
	IF pResult^.objectIdentifier = iObject.ObjectID THEN
		pPropList := pResult^.pData;
		WHILE pPropList <> 0 DO
			IF pPropList^.ePropID = ePropID THEN
				CopyRemoteData(iObject, ePropID, pData, nData, F_BACnet_EndOf(pPropList, SIZEOF(ST_BACnetRM_PropertyValueList)), pPropList^.nValueSize -  SIZEOF(DWORD));
				ProcessResult:=S_OK;
			END_IF
			pPropList := F_BACnet_NextListElem(pPropList, pPropList^.nEntrySize);
		END_WHILE
	END_IF
	
	IF pCovSlaves <> 0 AND nCovSlaves > 0 THEN
		FOR i:=0 TO nCovSlaves-1 DO
			pCovSlaves[i]^.ProcessResult(pResult);
		END_FOR
	END_IF
ELSE
	// (BETA) ... Output Error
END_IF
END_METHOD

METHOD PROTECTED StartTimer : BOOL
VAR_INPUT
END_VAR
timer(IN:=FALSE, PT:=tLifetime);
timer(IN:=TRUE, PT:=tLifetime);
END_METHOD

METHOD FB_Exit : BOOL
VAR_INPUT
	 bInCopyCode : BOOL; // if TRUE, the exit method is called for exiting an instance that is copied afterwards (online change).
END_VAR
VAR
	i : UDINT;
END_VAR
IF pCovSlaves <> 0 THEN
	__DELETE(pCovSlaves);
	pCovSlaves:=0;
END_IF
pMaster:=0;
END_METHOD

METHOD GetRequestType : E_BACnetRM_RequestType
VAR_INPUT
END_VAR
GetRequestType := E_BACnetRM_RequestType.eCov;
END_METHOD

METHOD IsReady : BOOL
VAR_INPUT
END_VAR
IF NOT bSendSubs THEN
	IsReady:=TRUE;
	RETURN;
END_IF

IsReady:=SUPER^.IsReady();
END_METHOD

PROPERTY Master : POINTER TO FB_BACnetRM_ReqCov
GET
Master:=pMaster;
END_GET
SET
pMaster:=Master;
END_SET
END_PROPERTY

PROPERTY SendSubscription : BOOL
GET
SendSubscription:=bSendSubs;
END_GET
SET
bSendSubs:=SendSubscription;
END_SET
END_PROPERTY

END_FUNCTION_BLOCK

// POUs/Remote/Objects/Basic/[Base]/FB_BACnetRM_BaseTLog
FUNCTION_BLOCK FB_BACnetRM_BaseTLog EXTENDS FB_BACnetRM_EventObject
VAR_OUTPUT
	nRecordCount				: UDINT;
	nTotalRecordCount			: UDINT;
END_VAR

SUPER^();

METHOD PROTECTED OnObjectStateChanged
SUPER^.OnObjectStateChanged();

SyncProperty(E_BACnetPropIdentifier.PropRecordCount, SIZEOF(nRecordCount), ADR(nRecordCount), E_BA_SyncModeRM.eRead);
SyncProperty(E_BACnetPropIdentifier.PropTotalRecordCount, SIZEOF(nTotalRecordCount), ADR(nTotalRecordCount), E_BA_SyncModeRM.eRead);
END_METHOD

END_FUNCTION_BLOCK

// POUs/Remote/Objects/Basic/[Base]/FB_BACnetRM_EventObject
FUNCTION_BLOCK FB_BACnetRM_EventObject EXTENDS FB_BACnetRM_Object
VAR_OUTPUT
	bEvent						: BOOL;												// Indicates an active event
END_VAR
VAR
	{region 'Event'}
		stStatusFlags			: ST_BA_StatusFlags;
	{endregion}
END_VAR

SUPER^();

bEvent := F_BA_IsDisturbed(stStatusFlags);

METHOD PROTECTED OnObjectStateChanged
SUPER^.OnObjectStateChanged();

SyncProperty(E_BACnetPropIdentifier.PropStatusFlags, SIZEOF(stStatusFlags), ADR(stStatusFlags), E_BA_SyncModeRM.eRead);
END_METHOD

PROPERTY StatusFlags : ST_BA_StatusFlags
GET
StatusFlags := stStatusFlags;
END_GET
END_PROPERTY

END_FUNCTION_BLOCK

// POUs/Remote/Objects/Basic/FB_BACnetRM_Acc
{attribute 'enable_dynamic_creation'}
FUNCTION_BLOCK FB_BACnetRM_Acc EXTENDS FB_BACnetRM_EventObject
VAR_OUTPUT
	nPresentValue			: UDINT;
END_VAR

SUPER^();

METHOD PROTECTED OnObjectStateChanged
SUPER^.OnObjectStateChanged();

SyncProperty(E_BACnetPropIdentifier.PropPresentValue, SIZEOF(nPresentValue), ADR(nPresentValue), E_BA_SyncModeRM.eRead);
END_METHOD

METHOD FB_init : BOOL
VAR_INPUT
	bInitRetains : BOOL; // if TRUE, the retain variables are initialized (warm start / cold start)
	bInCopyCode : BOOL;  // if TRUE, the instance afterwards gets moved into the copy code (online change)
END_VAR
eObjectType := E_BACnetObjType.ObjAccumulator;
END_METHOD

END_FUNCTION_BLOCK

// POUs/Remote/Objects/Basic/FB_BACnetRM_AI
{attribute 'enable_dynamic_creation'}
FUNCTION_BLOCK FB_BACnetRM_AI EXTENDS FB_BACnetRM_EventObject
VAR_INPUT CONSTANT PERSISTENT
	{region 'Fixed Parameters'}
		{attribute 'parameterCategory':='Config'}
		fReadIncrement : REAL; 
	{endregion}
END_VAR
VAR_OUTPUT
	fPresentValue 	: REAL;
END_VAR

SUPER^();

METHOD PROTECTED OnObjectStateChanged
SUPER^.OnObjectStateChanged();

SyncPropertyReal(E_BACnetPropIdentifier.PropPresentValue, SIZEOF(fPresentValue), ADR(fPresentValue), E_BA_SyncModeRM.eRead, fReadIncrement);
END_METHOD

METHOD FB_init : BOOL
VAR_INPUT
	bInitRetains : BOOL; // if TRUE, the retain variables are initialized (warm start / cold start)
	bInCopyCode : BOOL;  // if TRUE, the instance afterwards gets moved into the copy code (online change)
END_VAR
eObjectType := E_BACnetObjType.ObjAnalogInput;
END_METHOD

END_FUNCTION_BLOCK

// POUs/Remote/Objects/Basic/FB_BACnetRM_AO
{attribute 'enable_dynamic_creation'}
FUNCTION_BLOCK FB_BACnetRM_AO EXTENDS FB_BACnetRM_EventObject
VAR_INPUT
	fPv 			: REAL;
	bEnablePv 		: BOOL;
	bNullPv 		: BOOL;
END_VAR
VAR_INPUT CONSTANT PERSISTENT
	{region 'Fixed Parameters'}
		{attribute 'parameterCategory':='Config'}
		fReadIncrement : REAL; 
		{attribute 'parameterCategory':='Config'}
		fWriteIncrement : REAL; 
			 
		{attribute 'parameterCategory':='Value'}
		ePriority : E_BACnet_Priority := BACnet_Param.eRemotePrio_Default;
	{endregion}
END_VAR
VAR_OUTPUT
	fPresentValue 	: REAL;
END_VAR

SUPER^();

METHOD PROTECTED OnObjectStateChanged
SUPER^.OnObjectStateChanged();

SyncPropertyReal(E_BACnetPropIdentifier.PropPresentValue, SIZEOF(fPresentValue), ADR(fPresentValue), E_BA_SyncModeRM.eRead, fReadIncrement);

SyncPropertyPrioReal(E_BACnetPropIdentifier.PropPresentValue, SIZEOF(fPv), ADR(fPv), ADR(bEnablePv), ADR(bNullPv), ePriority, E_BA_SyncModeRM.eWrite, fWriteIncrement);
END_METHOD

METHOD FB_init : BOOL
VAR_INPUT
	bInitRetains : BOOL; // if TRUE, the retain variables are initialized (warm start / cold start)
	bInCopyCode : BOOL;  // if TRUE, the instance afterwards gets moved into the copy code (online change)
END_VAR
eObjectType := E_BACnetObjType.ObjAnalogOutput;
END_METHOD

END_FUNCTION_BLOCK

// POUs/Remote/Objects/Basic/FB_BACnetRM_AV
{attribute 'enable_dynamic_creation'}
FUNCTION_BLOCK FB_BACnetRM_AV EXTENDS FB_BACnetRM_EventObject
VAR_INPUT
	fPv 			: REAL;
	bEnablePv 		: BOOL;
	bNullPv 		: BOOL;	
END_VAR
VAR_INPUT CONSTANT PERSISTENT
	{region 'Fixed Parameters'}
		{attribute 'parameterCategory':='Config'}
		fReadIncrement : REAL; 
		{attribute 'parameterCategory':='Config'}
		fWriteIncrement : REAL; 
			 
		{attribute 'parameterCategory':='Value'}
		ePriority 	  : E_BACnet_Priority := BACnet_Param.eRemotePrio_Default;
	{endregion}
END_VAR
VAR_OUTPUT
	fPresentValue 	: REAL;
END_VAR

SUPER^();

METHOD PROTECTED OnObjectStateChanged
SUPER^.OnObjectStateChanged();

SyncPropertyReal(E_BACnetPropIdentifier.PropPresentValue, SIZEOF(fPresentValue), ADR(fPresentValue), E_BA_SyncModeRM.eRead, fReadIncrement);

SyncPropertyPrioReal(E_BACnetPropIdentifier.PropPresentValue, SIZEOF(fPv), ADR(fPv), ADR(bEnablePv), ADR(bNullPv), ePriority, E_BA_SyncModeRM.eWrite, fWriteIncrement);
END_METHOD

METHOD FB_init : BOOL
VAR_INPUT
	bInitRetains : BOOL; // if TRUE, the retain variables are initialized (warm start / cold start)
	bInCopyCode : BOOL;  // if TRUE, the instance afterwards gets moved into the copy code (online change)
END_VAR
eObjectType := E_BACnetObjType.ObjAnalogValue;
END_METHOD

END_FUNCTION_BLOCK

// POUs/Remote/Objects/Basic/FB_BACnetRM_AV_Disp
{attribute 'enable_dynamic_creation'}
FUNCTION_BLOCK FB_BACnetRM_AV_Disp EXTENDS FB_BACnetRM_Object
VAR_INPUT CONSTANT PERSISTENT
	{region 'Fixed Parameters'}
		{attribute 'parameterCategory':='Config'}
		fReadIncrement : REAL;
	{endregion}
END_VAR
VAR_OUTPUT
	fPresentValue 	: REAL;
END_VAR

SUPER^();

METHOD PROTECTED OnObjectStateChanged
SUPER^.OnObjectStateChanged();

SyncPropertyReal(E_BACnetPropIdentifier.PropPresentValue, SIZEOF(fPresentValue), ADR(fPresentValue), E_BA_SyncModeRM.eRead, fReadIncrement);
END_METHOD

METHOD FB_init : BOOL
VAR_INPUT
	bInitRetains : BOOL; // if TRUE, the retain variables are initialized (warm start / cold start)
	bInCopyCode : BOOL;  // if TRUE, the instance afterwards gets moved into the copy code (online change)
END_VAR
eObjectType := E_BACnetObjType.ObjAnalogValue;
END_METHOD

END_FUNCTION_BLOCK

// POUs/Remote/Objects/Basic/FB_BACnetRM_AV_Setp
{attribute 'enable_dynamic_creation'}
FUNCTION_BLOCK FB_BACnetRM_AV_Setp EXTENDS FB_BACnetRM_Object
VAR_INPUT CONSTANT PERSISTENT
	{region 'Fixed Parameters'}
		{attribute 'parameterCategory':='Config'}
		fReadIncrement : REAL; 
		{attribute 'parameterCategory':='Config'}
		fWriteIncrement : REAL; 
	{endregion}
END_VAR
VAR_INPUT CONSTANT
	{region 'Operational Parameters'}
		{attribute 'parameterCategory':='Value'}
		fValue : REAL;
	{endregion}
END_VAR
VAR_OUTPUT
	fPresentValue 	: REAL;
END_VAR

SUPER^();

{attribute 'hide'}
METHOD OnCOV
VAR_INPUT
	ePropID		: E_BACnetPropIdentifier;
END_VAR
CASE (ePropID) OF
	E_BACnetPropIdentifier.PropPresentValue:
		fValue := fPresentValue;
		
ELSE
	SUPER^.OnCOV(ePropID);
END_CASE
END_METHOD

METHOD PROTECTED OnObjectStateChanged
SUPER^.OnObjectStateChanged();

SyncPropertyReal(E_BACnetPropIdentifier.PropPresentValue, SIZEOF(fPresentValue), ADR(fPresentValue), E_BA_SyncModeRM.eRead, fReadIncrement);

SyncPropertyReal(E_BACnetPropIdentifier.PropPresentValue, SIZEOF(fValue), ADR(fValue), E_BA_SyncModeRM.eWrite, fWriteIncrement);
END_METHOD

METHOD FB_init : BOOL
VAR_INPUT
	bInitRetains : BOOL; // if TRUE, the retain variables are initialized (warm start / cold start)
	bInCopyCode : BOOL;  // if TRUE, the instance afterwards gets moved into the copy code (online change)
END_VAR
eObjectType := E_BACnetObjType.ObjAnalogValue;
END_METHOD

END_FUNCTION_BLOCK

// POUs/Remote/Objects/Basic/FB_BACnetRM_Avg
{attribute 'enable_dynamic_creation'}
FUNCTION_BLOCK FB_BACnetRM_Avg EXTENDS FB_BACnetRM_Object
VAR_OUTPUT
	fAverageValue			: REAL;
	fMinimumValue			: REAL;
	fMaximumValue			: REAL;
END_VAR

SUPER^();

METHOD PROTECTED OnObjectStateChanged
VAR
	nPresentValue: INT;
END_VAR
SUPER^.OnObjectStateChanged();

SyncProperty(E_BACnetPropIdentifier.PropAverageValue, SIZEOF(fAverageValue), ADR(fAverageValue), E_BA_SyncModeRM.eRead);
SyncProperty(E_BACnetPropIdentifier.PropMinimumValue, SIZEOF(fMinimumValue), ADR(fMinimumValue), E_BA_SyncModeRM.eRead);
SyncProperty(E_BACnetPropIdentifier.PropMaximumValue, SIZEOF(fMaximumValue), ADR(fMaximumValue), E_BA_SyncModeRM.eRead);
END_METHOD

METHOD FB_init : BOOL
VAR_INPUT
	bInitRetains : BOOL; // if TRUE, the retain variables are initialized (warm start / cold start)
	bInCopyCode : BOOL;  // if TRUE, the instance afterwards gets moved into the copy code (online change)
END_VAR
eObjectType := E_BACnetObjType.ObjAveraging;
END_METHOD

END_FUNCTION_BLOCK

// POUs/Remote/Objects/Basic/FB_BACnetRM_BI
{attribute 'enable_dynamic_creation'}
FUNCTION_BLOCK FB_BACnetRM_BI EXTENDS FB_BACnetRM_EventObject
VAR_OUTPUT
	bPresentValue 	: BOOL;
END_VAR

SUPER^();

METHOD PROTECTED OnObjectStateChanged
SUPER^.OnObjectStateChanged();

SyncProperty(E_BACnetPropIdentifier.PropPresentValue, SIZEOF(bPresentValue), ADR(bPresentValue), E_BA_SyncModeRM.eRead);
END_METHOD

METHOD FB_init : BOOL
VAR_INPUT
	bInitRetains : BOOL; // if TRUE, the retain variables are initialized (warm start / cold start)
	bInCopyCode : BOOL;  // if TRUE, the instance afterwards gets moved into the copy code (online change)
END_VAR
eObjectType := E_BACnetObjType.ObjBinaryInput;
END_METHOD

END_FUNCTION_BLOCK

// POUs/Remote/Objects/Basic/FB_BACnetRM_BO
{attribute 'enable_dynamic_creation'}
FUNCTION_BLOCK FB_BACnetRM_BO EXTENDS FB_BACnetRM_EventObject
VAR_INPUT
	bPv 			: BOOL;
	bEnablePv 		: BOOL;
	bNullPv 		: BOOL;	
END_VAR
VAR_INPUT CONSTANT PERSISTENT
	{region 'Fixed Parameters'}
		{attribute 'parameterCategory':='Value'}
		ePriority : E_BACnet_Priority := BACnet_Param.eRemotePrio_Default;
	{endregion}
END_VAR
VAR_OUTPUT
	bPresentValue 	: BOOL;
END_VAR

SUPER^();

METHOD PROTECTED OnObjectStateChanged
SUPER^.OnObjectStateChanged();

SyncProperty(E_BACnetPropIdentifier.PropPresentValue, SIZEOF(bPresentValue), ADR(bPresentValue), E_BA_SyncModeRM.eRead);

SyncPropertyPrio(E_BACnetPropIdentifier.PropPresentValue, SIZEOF(bPv), ADR(bPv), ADR(bEnablePv), ADR(bNullPv), ePriority, E_BA_SyncModeRM.eWrite);
END_METHOD

METHOD FB_init : BOOL
VAR_INPUT
	bInitRetains : BOOL; // if TRUE, the retain variables are initialized (warm start / cold start)
	bInCopyCode : BOOL;  // if TRUE, the instance afterwards gets moved into the copy code (online change)
END_VAR
eObjectType := E_BACnetObjType.ObjBinaryOutput;
END_METHOD

END_FUNCTION_BLOCK

// POUs/Remote/Objects/Basic/FB_BACnetRM_BV
{attribute 'enable_dynamic_creation'}
FUNCTION_BLOCK FB_BACnetRM_BV EXTENDS FB_BACnetRM_EventObject
VAR_INPUT
	bPv 			: BOOL;
	bEnablePv 		: BOOL;
	bNullPv 		: BOOL;	
END_VAR
VAR_INPUT CONSTANT PERSISTENT
	{region 'Fixed Parameters'}
		{attribute 'parameterCategory':='Value'}
		ePriority : E_BACnet_Priority := BACnet_Param.eRemotePrio_Default;
	{endregion}
END_VAR
VAR_OUTPUT
	bPresentValue 	: BOOL;
END_VAR

SUPER^();

METHOD PROTECTED OnObjectStateChanged
SUPER^.OnObjectStateChanged();

SyncProperty(E_BACnetPropIdentifier.PropPresentValue, SIZEOF(bPresentValue), ADR(bPresentValue), E_BA_SyncModeRM.eRead);

SyncPropertyPrio(E_BACnetPropIdentifier.PropPresentValue, SIZEOF(bPv), ADR(bPv), ADR(bEnablePv), ADR(bNullPv), ePriority, E_BA_SyncModeRM.eWrite);
END_METHOD

METHOD FB_init : BOOL
VAR_INPUT
	bInitRetains : BOOL; // if TRUE, the retain variables are initialized (warm start / cold start)
	bInCopyCode : BOOL;  // if TRUE, the instance afterwards gets moved into the copy code (online change)
END_VAR
eObjectType := E_BACnetObjType.ObjBinaryValue;
END_METHOD

END_FUNCTION_BLOCK

// POUs/Remote/Objects/Basic/FB_BACnetRM_BV_Disp
{attribute 'enable_dynamic_creation'}
FUNCTION_BLOCK FB_BACnetRM_BV_Disp EXTENDS FB_BACnetRM_Object
VAR_OUTPUT
	bPresentValue	: BOOL;
END_VAR

SUPER^();

METHOD PROTECTED OnObjectStateChanged
SUPER^.OnObjectStateChanged();

SyncProperty(E_BACnetPropIdentifier.PropPresentValue, SIZEOF(bPresentValue), ADR(bPresentValue), E_BA_SyncModeRM.eRead);
END_METHOD

METHOD FB_init : BOOL
VAR_INPUT
	bInitRetains : BOOL; // if TRUE, the retain variables are initialized (warm start / cold start)
	bInCopyCode : BOOL;  // if TRUE, the instance afterwards gets moved into the copy code (online change)
END_VAR
eObjectType := E_BACnetObjType.ObjBinaryValue;
END_METHOD

END_FUNCTION_BLOCK

// POUs/Remote/Objects/Basic/FB_BACnetRM_BV_Setp
{attribute 'enable_dynamic_creation'}
FUNCTION_BLOCK FB_BACnetRM_BV_Setp EXTENDS FB_BACnetRM_Object
VAR_INPUT CONSTANT
	{region 'Operational Parameters'}
		{attribute 'parameterCategory':='Value'}
		bValue : BOOL;
	{endregion}
END_VAR
VAR_OUTPUT
	bPresentValue	: BOOL;
END_VAR

SUPER^();

{attribute 'hide'}
METHOD OnCOV
VAR_INPUT
	ePropID		: E_BACnetPropIdentifier;
END_VAR
CASE (ePropID) OF
	E_BACnetPropIdentifier.PropPresentValue:
		bValue := bPresentValue;
		
ELSE
	SUPER^.OnCOV(ePropID);
END_CASE
END_METHOD

METHOD PROTECTED OnObjectStateChanged
SUPER^.OnObjectStateChanged();

SyncProperty(E_BACnetPropIdentifier.PropPresentValue, SIZEOF(bPresentValue), ADR(bPresentValue), E_BA_SyncModeRM.eRead);

SyncProperty(E_BACnetPropIdentifier.PropPresentValue, SIZEOF(bValue), ADR(bValue), E_BA_SyncModeRM.eWrite);
END_METHOD

METHOD FB_init : BOOL
VAR_INPUT
	bInitRetains : BOOL; // if TRUE, the retain variables are initialized (warm start / cold start)
	bInCopyCode : BOOL;  // if TRUE, the instance afterwards gets moved into the copy code (online change)
END_VAR
eObjectType := E_BACnetObjType.ObjBinaryValue;
END_METHOD

END_FUNCTION_BLOCK

// POUs/Remote/Objects/Basic/FB_BACnetRM_Cal
{attribute 'enable_dynamic_creation'}
FUNCTION_BLOCK FB_BACnetRM_Cal EXTENDS FB_BACnetRM_Object
VAR_OUTPUT
	bPresentValue 	: BOOL;
END_VAR

SUPER^();

METHOD PROTECTED OnObjectStateChanged
SUPER^.OnObjectStateChanged();

SyncProperty(E_BACnetPropIdentifier.PropPresentValue, SIZEOF(bPresentValue), ADR(bPresentValue), E_BA_SyncModeRM.eRead);
END_METHOD

METHOD FB_init : BOOL
VAR_INPUT
	bInitRetains : BOOL; // if TRUE, the retain variables are initialized (warm start / cold start)
	bInCopyCode : BOOL;  // if TRUE, the instance afterwards gets moved into the copy code (online change)
END_VAR
eObjectType := E_BACnetObjType.ObjCalendar;
END_METHOD

END_FUNCTION_BLOCK

// POUs/Remote/Objects/Basic/FB_BACnetRM_Cmd
{attribute 'enable_dynamic_creation'}
FUNCTION_BLOCK FB_BACnetRM_Cmd EXTENDS FB_BACnetRM_Object
VAR_OUTPUT
	nPresentValue		: UDINT;
	bAllWritesOk		: BOOL; (* all actions in selected action list are written *)
	bInProcess			: BOOL; (* object is busy *)
END_VAR

SUPER^();

METHOD PROTECTED OnObjectStateChanged
SUPER^.OnObjectStateChanged();

SyncProperty(E_BACnetPropIdentifier.PropPresentValue, SIZEOF(nPresentValue), ADR(nPresentValue), E_BA_SyncModeRM.eRead);
SyncProperty(E_BACnetPropIdentifier.PropAllWritesSuccessful, SIZEOF(bAllWritesOk), ADR(bAllWritesOk), E_BA_SyncModeRM.eRead);
SyncProperty(E_BACnetPropIdentifier.PropInProcess, SIZEOF(bInProcess), ADR(bInProcess), E_BA_SyncModeRM.eRead);
END_METHOD

METHOD FB_init : BOOL
VAR_INPUT
	bInitRetains : BOOL; // if TRUE, the retain variables are initialized (warm start / cold start)
	bInCopyCode : BOOL;  // if TRUE, the instance afterwards gets moved into the copy code (online change)
END_VAR
eObjectType := E_BACnetObjType.ObjCommand;
END_METHOD

END_FUNCTION_BLOCK

// POUs/Remote/Objects/Basic/FB_BACnetRM_Device
{attribute 'enable_dynamic_creation'}
FUNCTION_BLOCK FB_BACnetRM_Device EXTENDS FB_BACnetRM_Object
VAR_OUTPUT
	bOperational		: BOOL;
END_VAR

IF (NOT bReady) THEN
	IF (nObjectInstance = BACnet_Globals.nBACnetInstId_Auto) THEN
		nObjectInstance:=Client.ObjectInstance;
	END_IF
END_IF

SUPER^();

METHOD PROTECTED OnObjectStateChanged
SUPER^.OnObjectStateChanged();

IF (nObjectInstance = 16#23FFFFF) THEN
	nObjectInstance := Client.ObjectInstance;
END_IF

SyncProperty(E_BACnetPropIdentifier.PropSystemStatus, SIZEOF(bOperational), ADR(bOperational), E_BA_SyncModeRM.eRead);
END_METHOD

METHOD FB_init : BOOL
VAR_INPUT
	bInitRetains : BOOL; // if TRUE, the retain variables are initialized (warm start / cold start)
	bInCopyCode : BOOL;  // if TRUE, the instance afterwards gets moved into the copy code (online change)
END_VAR
eObjectType := E_BACnetObjType.ObjDevice;
END_METHOD

END_FUNCTION_BLOCK

// POUs/Remote/Objects/Basic/FB_BACnetRM_EE
{attribute 'enable_dynamic_creation'}
FUNCTION_BLOCK FB_BACnetRM_EE EXTENDS FB_BACnetRM_Object
VAR_OUTPUT
END_VAR

SUPER^();

METHOD PROTECTED OnObjectStateChanged
SUPER^.OnObjectStateChanged();
END_METHOD

METHOD FB_init : BOOL
VAR_INPUT
	bInitRetains : BOOL; // if TRUE, the retain variables are initialized (warm start / cold start)
	bInCopyCode : BOOL;  // if TRUE, the instance afterwards gets moved into the copy code (online change)
END_VAR
eObjectType := E_BACnetObjType.ObjEventEnrollment;
END_METHOD

END_FUNCTION_BLOCK

// POUs/Remote/Objects/Basic/FB_BACnetRM_ELog
{attribute 'enable_dynamic_creation'}
FUNCTION_BLOCK FB_BACnetRM_ELog EXTENDS FB_BACnetRM_BaseTLog

SUPER^();

METHOD FB_init : BOOL
VAR_INPUT
	bInitRetains : BOOL; // if TRUE, the retain variables are initialized (warm start / cold start)
	bInCopyCode : BOOL;  // if TRUE, the instance afterwards gets moved into the copy code (online change)
END_VAR
eObjectType := E_BACnetObjType.ObjEventLog;
END_METHOD

END_FUNCTION_BLOCK

// POUs/Remote/Objects/Basic/FB_BACnetRM_File
{attribute 'enable_dynamic_creation'}
FUNCTION_BLOCK FB_BACnetRM_File EXTENDS FB_BACnetRM_Object
VAR_OUTPUT
	nFileSize		: UDINT;
END_VAR

SUPER^();

METHOD PROTECTED OnObjectStateChanged
SUPER^.OnObjectStateChanged();

SyncProperty(E_BACnetPropIdentifier.PropFileSize, SIZEOF(nFileSize), ADR(nFileSize), E_BA_SyncModeRM.eRead);
END_METHOD

METHOD FB_init : BOOL
VAR_INPUT
	bInitRetains : BOOL; // if TRUE, the retain variables are initialized (warm start / cold start)
	bInCopyCode : BOOL;  // if TRUE, the instance afterwards gets moved into the copy code (online change)
END_VAR
eObjectType := E_BACnetObjType.ObjFile;
END_METHOD

END_FUNCTION_BLOCK

// POUs/Remote/Objects/Basic/FB_BACnetRM_Group
{attribute 'enable_dynamic_creation'}
FUNCTION_BLOCK FB_BACnetRM_Group EXTENDS FB_BACnetRM_Object
VAR_OUTPUT
END_VAR

SUPER^();

METHOD PROTECTED OnObjectStateChanged
SUPER^.OnObjectStateChanged();
END_METHOD

METHOD FB_init : BOOL
VAR_INPUT
	bInitRetains : BOOL; // if TRUE, the retain variables are initialized (warm start / cold start)
	bInCopyCode : BOOL;  // if TRUE, the instance afterwards gets moved into the copy code (online change)
END_VAR
eObjectType := E_BACnetObjType.ObjGroup;
END_METHOD

END_FUNCTION_BLOCK

// POUs/Remote/Objects/Basic/FB_BACnetRM_Loop
{attribute 'enable_dynamic_creation'}
FUNCTION_BLOCK FB_BACnetRM_Loop EXTENDS FB_BACnetRM_EventObject
VAR_OUTPUT
	fPresentValue		: REAL;
	fSetpoint			: REAL;
	fCtrlVar			: REAL;
END_VAR

SUPER^();

METHOD PROTECTED OnObjectStateChanged
SUPER^.OnObjectStateChanged();

SyncProperty(E_BACnetPropIdentifier.PropPresentValue, SIZEOF(fPresentValue), ADR(fPresentValue), E_BA_SyncModeRM.eRead);
SyncProperty(E_BACnetPropIdentifier.PropSetpoint, SIZEOF(fSetpoint), ADR(fSetpoint), E_BA_SyncModeRM.eRead);
SyncProperty(E_BACnetPropIdentifier.PropControlledVariableValue, SIZEOF(fCtrlVar), ADR(fCtrlVar), E_BA_SyncModeRM.eRead);
END_METHOD

METHOD FB_init : BOOL
VAR_INPUT
	bInitRetains : BOOL; // if TRUE, the retain variables are initialized (warm start / cold start)
	bInCopyCode : BOOL;  // if TRUE, the instance afterwards gets moved into the copy code (online change)
END_VAR
eObjectType := E_BACnetObjType.ObjLoop;
END_METHOD

END_FUNCTION_BLOCK

// POUs/Remote/Objects/Basic/FB_BACnetRM_MI
{attribute 'enable_dynamic_creation'}
FUNCTION_BLOCK FB_BACnetRM_MI EXTENDS FB_BACnetRM_EventObject
VAR_OUTPUT
	nPresentValue 	: UDINT;
END_VAR

SUPER^();

METHOD PROTECTED OnObjectStateChanged
SUPER^.OnObjectStateChanged();

SyncProperty(E_BACnetPropIdentifier.PropPresentValue, SIZEOF(nPresentValue), ADR(nPresentValue), E_BA_SyncModeRM.eRead);
END_METHOD

METHOD FB_init : BOOL
VAR_INPUT
	bInitRetains : BOOL; // if TRUE, the retain variables are initialized (warm start / cold start)
	bInCopyCode : BOOL;  // if TRUE, the instance afterwards gets moved into the copy code (online change)
END_VAR
eObjectType := E_BACnetObjType.ObjMultistateInput;
END_METHOD

END_FUNCTION_BLOCK

// POUs/Remote/Objects/Basic/FB_BACnetRM_MO
{attribute 'enable_dynamic_creation'}
FUNCTION_BLOCK FB_BACnetRM_MO EXTENDS FB_BACnetRM_EventObject
VAR_INPUT
	nPv 			: UDINT;
	bEnablePv 		: BOOL;
	bNullPv 		: BOOL;	
END_VAR
VAR_INPUT CONSTANT PERSISTENT
	{region 'Fixed Parameters'}
		{attribute 'parameterCategory':='Value'}
		ePriority : E_BACnet_Priority := BACnet_Param.eRemotePrio_Default;
	{endregion}
END_VAR
VAR_OUTPUT
	nPresentValue 	: UDINT;
END_VAR

SUPER^();

METHOD PROTECTED OnObjectStateChanged
SUPER^.OnObjectStateChanged();

SyncProperty(E_BACnetPropIdentifier.PropPresentValue, SIZEOF(nPresentValue), ADR(nPresentValue), E_BA_SyncModeRM.eRead);

SyncPropertyPrio(E_BACnetPropIdentifier.PropPresentValue, SIZEOF(nPv), ADR(nPv), ADR(bEnablePv), ADR(bNullPv), ePriority, E_BA_SyncModeRM.eWrite);
END_METHOD

METHOD FB_init : BOOL
VAR_INPUT
	bInitRetains : BOOL; // if TRUE, the retain variables are initialized (warm start / cold start)
	bInCopyCode : BOOL;  // if TRUE, the instance afterwards gets moved into the copy code (online change)
END_VAR
eObjectType := E_BACnetObjType.ObjMultistateOutput;
END_METHOD

END_FUNCTION_BLOCK

// POUs/Remote/Objects/Basic/FB_BACnetRM_MV
{attribute 'enable_dynamic_creation'}
FUNCTION_BLOCK FB_BACnetRM_MV EXTENDS FB_BACnetRM_EventObject
VAR_INPUT
	nPv 			: UDINT;
	bEnablePv 		: BOOL;
	bNullPv 		: BOOL;	
END_VAR
VAR_INPUT CONSTANT PERSISTENT
	{region 'Fixed Parameters'}
		{attribute 'parameterCategory':='Value'}
		ePriority : E_BACnet_Priority := BACnet_Param.eRemotePrio_Default;
	{endregion}
END_VAR
VAR_OUTPUT
	nPresentValue 	: UDINT;
END_VAR

SUPER^();

METHOD PROTECTED OnObjectStateChanged
SUPER^.OnObjectStateChanged();

SyncProperty(E_BACnetPropIdentifier.PropPresentValue, SIZEOF(nPresentValue), ADR(nPresentValue), E_BA_SyncModeRM.eRead);

SyncPropertyPrio(E_BACnetPropIdentifier.PropPresentValue, SIZEOF(nPv), ADR(nPv), ADR(bEnablePv), ADR(bNullPv), ePriority, E_BA_SyncModeRM.eWrite);
END_METHOD

METHOD FB_init : BOOL
VAR_INPUT
	bInitRetains : BOOL; // if TRUE, the retain variables are initialized (warm start / cold start)
	bInCopyCode : BOOL;  // if TRUE, the instance afterwards gets moved into the copy code (online change)
END_VAR
eObjectType := E_BACnetObjType.ObjMultistateValue;
END_METHOD

END_FUNCTION_BLOCK

// POUs/Remote/Objects/Basic/FB_BACnetRM_MV_Disp
{attribute 'enable_dynamic_creation'}
FUNCTION_BLOCK FB_BACnetRM_MV_Disp EXTENDS FB_BACnetRM_Object
VAR_OUTPUT
	nPresentValue		: UDINT		:= 1;
END_VAR

SUPER^();

METHOD PROTECTED OnObjectStateChanged
SUPER^.OnObjectStateChanged();

SyncProperty(E_BACnetPropIdentifier.PropPresentValue, SIZEOF(nPresentValue), ADR(nPresentValue), E_BA_SyncModeRM.eRead);
END_METHOD

METHOD FB_init : BOOL
VAR_INPUT
	bInitRetains : BOOL; // if TRUE, the retain variables are initialized (warm start / cold start)
	bInCopyCode : BOOL;  // if TRUE, the instance afterwards gets moved into the copy code (online change)
END_VAR
eObjectType := E_BACnetObjType.ObjMultistateValue;
END_METHOD

END_FUNCTION_BLOCK

// POUs/Remote/Objects/Basic/FB_BACnetRM_MV_Setp
{attribute 'enable_dynamic_creation'}
FUNCTION_BLOCK FB_BACnetRM_MV_Setp EXTENDS FB_BACnetRM_Object
VAR_INPUT CONSTANT
	{region 'Operational Parameters'}
		{attribute 'parameterCategory':='Value'}
		nValue : UDINT;
	{endregion}
END_VAR
VAR_OUTPUT
	nPresentValue		: UDINT		:= 1;
END_VAR

SUPER^();

{attribute 'hide'}
METHOD OnCOV
VAR_INPUT
	ePropID		: E_BACnetPropIdentifier;
END_VAR
CASE (ePropID) OF
	E_BACnetPropIdentifier.PropPresentValue:
		nValue := nPresentValue;
		
ELSE
	SUPER^.OnCOV(ePropID);
END_CASE
END_METHOD

METHOD PROTECTED OnObjectStateChanged
SUPER^.OnObjectStateChanged();

SyncProperty(E_BACnetPropIdentifier.PropPresentValue, SIZEOF(nPresentValue), ADR(nPresentValue), E_BA_SyncModeRM.eRead);

SyncProperty(E_BACnetPropIdentifier.PropPresentValue, SIZEOF(nValue), ADR(nValue), E_BA_SyncModeRM.eWrite);
END_METHOD

METHOD FB_init : BOOL
VAR_INPUT
	bInitRetains : BOOL; // if TRUE, the retain variables are initialized (warm start / cold start)
	bInCopyCode : BOOL;  // if TRUE, the instance afterwards gets moved into the copy code (online change)
END_VAR
eObjectType := E_BACnetObjType.ObjMultistateValue;
END_METHOD

END_FUNCTION_BLOCK

// POUs/Remote/Objects/Basic/FB_BACnetRM_NC
{attribute 'enable_dynamic_creation'}
FUNCTION_BLOCK FB_BACnetRM_NC EXTENDS FB_BACnetRM_Object
VAR_OUTPUT
	nNotificationClass		: UDINT;
END_VAR

SUPER^();

METHOD PROTECTED OnObjectStateChanged
SUPER^.OnObjectStateChanged();

SyncProperty(E_BACnetPropIdentifier.PropNotificationClass, SIZEOF(nNotificationClass), ADR(nNotificationClass), E_BA_SyncModeRM.eRead);
END_METHOD

METHOD FB_init : BOOL
VAR_INPUT
	bInitRetains : BOOL; // if TRUE, the retain variables are initialized (warm start / cold start)
	bInCopyCode : BOOL;  // if TRUE, the instance afterwards gets moved into the copy code (online change)
END_VAR
eObjectType := E_BACnetObjType.ObjNotificationClass;
END_METHOD

END_FUNCTION_BLOCK

// POUs/Remote/Objects/Basic/FB_BACnetRM_PC
{attribute 'enable_dynamic_creation'}
FUNCTION_BLOCK FB_BACnetRM_PC EXTENDS FB_BACnetRM_EventObject
VAR_OUTPUT
	fPresentValue			: REAL;
END_VAR

SUPER^();

METHOD PROTECTED OnObjectStateChanged
SUPER^.OnObjectStateChanged();

SyncProperty(E_BACnetPropIdentifier.PropPresentValue, SIZEOF(fPresentValue), ADR(fPresentValue), E_BA_SyncModeRM.eRead);
END_METHOD

METHOD FB_init : BOOL
VAR_INPUT
	bInitRetains : BOOL; // if TRUE, the retain variables are initialized (warm start / cold start)
	bInCopyCode : BOOL;  // if TRUE, the instance afterwards gets moved into the copy code (online change)
END_VAR
eObjectType := E_BACnetObjType.ObjPulseConverter;
END_METHOD

END_FUNCTION_BLOCK

// POUs/Remote/Objects/Basic/FB_BACnetRM_Prog
{attribute 'enable_dynamic_creation'}
FUNCTION_BLOCK FB_BACnetRM_Prog EXTENDS FB_BACnetRM_EventObject
VAR_OUTPUT
	eState			: E_BACnet_ProgramState;
END_VAR

SUPER^();

METHOD PROTECTED OnObjectStateChanged
SUPER^.OnObjectStateChanged();

SyncProperty(E_BACnetPropIdentifier.PropProgramState, SIZEOF(eState), ADR(eState), E_BA_SyncModeRM.eRead);
END_METHOD

METHOD FB_init : BOOL
VAR_INPUT
	bInitRetains : BOOL; // if TRUE, the retain variables are initialized (warm start / cold start)
	bInCopyCode : BOOL;  // if TRUE, the instance afterwards gets moved into the copy code (online change)
END_VAR
eObjectType := E_BACnetObjType.ObjProg;
END_METHOD

END_FUNCTION_BLOCK

// POUs/Remote/Objects/Basic/FB_BACnetRM_SchedA
{attribute 'enable_dynamic_creation'}
FUNCTION_BLOCK FB_BACnetRM_SchedA EXTENDS FB_BACnetRM_Object
VAR_OUTPUT
	fPresentValue 	: REAL;
END_VAR

SUPER^();

METHOD PROTECTED OnObjectStateChanged
SUPER^.OnObjectStateChanged();

SyncProperty(E_BACnetPropIdentifier.PropPresentValue, SIZEOF(fPresentValue), ADR(fPresentValue), E_BA_SyncModeRM.eRead);
END_METHOD

METHOD FB_init : BOOL
VAR_INPUT
	bInitRetains : BOOL; // if TRUE, the retain variables are initialized (warm start / cold start)
	bInCopyCode : BOOL;  // if TRUE, the instance afterwards gets moved into the copy code (online change)
END_VAR
eObjectType := E_BACnetObjType.ObjSchedule;
END_METHOD

END_FUNCTION_BLOCK

// POUs/Remote/Objects/Basic/FB_BACnetRM_SchedB
{attribute 'enable_dynamic_creation'}
FUNCTION_BLOCK FB_BACnetRM_SchedB EXTENDS FB_BACnetRM_Object
VAR_OUTPUT
	bPresentValue 	: BOOL;
END_VAR

SUPER^();

METHOD PROTECTED OnObjectStateChanged
SUPER^.OnObjectStateChanged();

SyncProperty(E_BACnetPropIdentifier.PropPresentValue, SIZEOF(bPresentValue), ADR(bPresentValue), E_BA_SyncModeRM.eRead);
END_METHOD

METHOD FB_init : BOOL
VAR_INPUT
	bInitRetains : BOOL; // if TRUE, the retain variables are initialized (warm start / cold start)
	bInCopyCode : BOOL;  // if TRUE, the instance afterwards gets moved into the copy code (online change)
END_VAR
eObjectType := E_BACnetObjType.ObjSchedule;
END_METHOD

END_FUNCTION_BLOCK

// POUs/Remote/Objects/Basic/FB_BACnetRM_SchedM
{attribute 'enable_dynamic_creation'}
FUNCTION_BLOCK FB_BACnetRM_SchedM EXTENDS FB_BACnetRM_Object
VAR_OUTPUT
	nPresentValue 	: UDINT;
END_VAR

SUPER^();

METHOD PROTECTED OnObjectStateChanged
SUPER^.OnObjectStateChanged();

SyncProperty(E_BACnetPropIdentifier.PropPresentValue, SIZEOF(nPresentValue), ADR(nPresentValue), E_BA_SyncModeRM.eRead);
END_METHOD

METHOD FB_init : BOOL
VAR_INPUT
	bInitRetains : BOOL; // if TRUE, the retain variables are initialized (warm start / cold start)
	bInCopyCode : BOOL;  // if TRUE, the instance afterwards gets moved into the copy code (online change)
END_VAR
eObjectType := E_BACnetObjType.ObjSchedule;
END_METHOD

END_FUNCTION_BLOCK

// POUs/Remote/Objects/Basic/FB_BACnetRM_TLM
{attribute 'enable_dynamic_creation'}
FUNCTION_BLOCK FB_BACnetRM_TLM EXTENDS FB_BACnetRM_BaseTLog

SUPER^();

METHOD FB_init : BOOL
VAR_INPUT
	bInitRetains : BOOL; // if TRUE, the retain variables are initialized (warm start / cold start)
	bInCopyCode : BOOL;  // if TRUE, the instance afterwards gets moved into the copy code (online change)
END_VAR
eObjectType := E_BACnetObjType.ObjTrendLogMultiple;
END_METHOD

END_FUNCTION_BLOCK

// POUs/Remote/Objects/Basic/FB_BACnetRM_TLog
{attribute 'enable_dynamic_creation'}
FUNCTION_BLOCK FB_BACnetRM_TLog EXTENDS FB_BACnetRM_BaseTLog

SUPER^();

METHOD FB_init : BOOL
VAR_INPUT
	bInitRetains : BOOL; // if TRUE, the retain variables are initialized (warm start / cold start)
	bInCopyCode : BOOL;  // if TRUE, the instance afterwards gets moved into the copy code (online change)
END_VAR
eObjectType := E_BACnetObjType.ObjTrendLog;
END_METHOD

END_FUNCTION_BLOCK

// POUs/Remote/Objects/Convenience/FB_BACnetRM_CnvLoop
{attribute 'enable_dynamic_creation'}
FUNCTION_BLOCK FB_BACnetRM_CnvLoop EXTENDS FB_BACnetRM_Loop
VAR_INPUT CONSTANT PERSISTENT
	{region 'Variable Parameters'}
		{attribute 'parameterCategory':='Config'}
		fPropertionalConstant : REAL;
		{attribute 'parameterCategory':='Config'}
		ePropertionalConstantUnit : E_BA_Unit;
		{attribute 'parameterCategory':='Config'}
		fIntegralConstant : REAL;
		{attribute 'parameterCategory':='Config'}
		eIntegralConstantUnit : E_BA_Unit;
		{attribute 'parameterCategory':='Config'}
		fDerivativeConstant : REAL;
		{attribute 'parameterCategory':='Config'}
		eDerivativeConstantUnit : E_BA_Unit;
	{endregion}
END_VAR

SUPER^();

METHOD PROTECTED OnObjectStateChanged
SUPER^.OnObjectStateChanged();

SyncProperty(E_BACnetPropIdentifier.PropProportionalConstant, SIZEOF(fPropertionalConstant), ADR(fPropertionalConstant), E_BA_SyncModeRM.eRead);
SyncProperty(E_BACnetPropIdentifier.PropProportionalConstantUnits, SIZEOF(ePropertionalConstantUnit), ADR(ePropertionalConstantUnit), E_BA_SyncModeRM.eRead);
SyncProperty(E_BACnetPropIdentifier.PropIntegralConstant, SIZEOF(fIntegralConstant), ADR(fIntegralConstant), E_BA_SyncModeRM.eRead);
SyncProperty(E_BACnetPropIdentifier.PropIntegralConstantUnits, SIZEOF(eIntegralConstantUnit), ADR(eIntegralConstantUnit), E_BA_SyncModeRM.eRead);
SyncProperty(E_BACnetPropIdentifier.PropDerivativeConstant, SIZEOF(fDerivativeConstant), ADR(fDerivativeConstant), E_BA_SyncModeRM.eRead);
SyncProperty(E_BACnetPropIdentifier.PropDerivativeConstantUnits, SIZEOF(eDerivativeConstantUnit), ADR(eDerivativeConstantUnit), E_BA_SyncModeRM.eRead);
END_METHOD

END_FUNCTION_BLOCK

// POUs/Remote/Objects/Experimental/FB_BACnetRM_ExpAV01
{attribute 'enable_dynamic_creation'}
{attribute 'hide'}	// (BETA) ...FB is only for testing!
FUNCTION_BLOCK FB_BACnetRM_ExpAV01 EXTENDS FB_BACnetRM_AV
VAR
	{region 'Test Properties'}
//		bHighLimitEnable		: BOOL;
//		fHighLimitValue			: REAL;
//		bLowLimitEnable			: BOOL;
//		fLowLimitValue			: REAL;
			 
		bWriteEnable			: BOOL;
		stLimitEnable 			: ST_BACnet_LimitEnableBits;
		stEventEnable 			: ST_BACnet_EventTransitionBits;		  
					   
		eReliability			: E_BA_Reliability;
		stAckedTransitions		: ST_BA_EventTransitions;
		eEventState				: E_BACnet_EventState;
	{endregion}
END_VAR

SUPER^();

METHOD PROTECTED OnObjectStateChanged
SUPER^.OnObjectStateChanged();

SyncProperty(E_BACnetPropIdentifier.PropReliability, SIZEOF(eReliability), ADR(eReliability), E_BA_SyncModeRM.eRead);
SyncProperty(E_BACnetPropIdentifier.PropEventState, SIZEOF(eEventState), ADR(eEventState), E_BA_SyncModeRM.eRead);
SyncProperty(E_BACnetPropIdentifier.PropAckedTransitions, SIZEOF(stAckedTransitions), ADR(stAckedTransitions), E_BA_SyncModeRM.eRead);


SyncPropertyEnable(E_BACnetPropIdentifier.PropEventEnable, SIZEOF(stEventEnable), ADR(stEventEnable), ADR(bWriteEnable), E_BA_SyncModeRM.eWrite);
SyncPropertyEnable(E_BACnetPropIdentifier.PropLimitEnable, SIZEOF(stLimitEnable), ADR(stLimitEnable), ADR(bWriteEnable), E_BA_SyncModeRM.eWrite);
END_METHOD

END_FUNCTION_BLOCK

// POUs/Remote/Objects/Experimental/FB_BACnetRM_ExpAV02
{attribute 'enable_dynamic_creation'}
{attribute 'hide'}	// (BETA) ...FB is only for testing!
FUNCTION_BLOCK FB_BACnetRM_ExpAV02 EXTENDS FB_BACnetRM_AV
VAR
	{region 'Test Properties'}
		stLimitEnable 			: ST_BACnet_LimitEnableBits;
	{endregion}
END_VAR
VAR
	{attribute 'hide'}
	fbLmEnWrite					: FB_BACnetRM_WriteProperty		:= (pData:=ADR(stLimitEnable), nData:=SIZEOF(stLimitEnable), ePropID:=PropLimitEnable, iObject:=THIS^);
	{attribute 'hide'}
	fbLmEnTrig					: FB_BA_ATrigCOV;
END_VAR

SUPER^();

IF (Client.bReady) THEN
	fbLmEnTrig(xValue:=stLimitEnable);
	fbLmEnWrite(Client:=Client, bExecute:=fbLmEnTrig.bQ);
END_IF

END_FUNCTION_BLOCK

// POUs/Remote/Objects/Primitive/FB_BACnetRM_BitString
{attribute 'enable_dynamic_creation'}
FUNCTION_BLOCK FB_BACnetRM_BitString EXTENDS FB_BACnetRM_Object
VAR_OUTPUT
	nPresentValue 	: ULINT;
END_VAR

SUPER^();

METHOD PROTECTED OnObjectStateChanged
SUPER^.OnObjectStateChanged();

SyncProperty(E_BACnetPropIdentifier.PropPresentValue, SIZEOF(nPresentValue), ADR(nPresentValue), E_BA_SyncModeRM.eRead);
END_METHOD

METHOD FB_init : BOOL
VAR_INPUT
	bInitRetains : BOOL; // if TRUE, the retain variables are initialized (warm start / cold start)
	bInCopyCode : BOOL;  // if TRUE, the instance afterwards gets moved into the copy code (online change)
END_VAR
eObjectType := E_BACnetObjType.ObjBitStringValue;
END_METHOD

END_FUNCTION_BLOCK

// POUs/Remote/Objects/Primitive/FB_BACnetRM_ByteArr
{attribute 'enable_dynamic_creation'}
FUNCTION_BLOCK FB_BACnetRM_ByteArr EXTENDS FB_BACnetRM_Object
VAR_OUTPUT
	aPresentValue 		: ARRAY [0..255] OF BYTE;
	nPresentValue 		: UINT;
END_VAR

SUPER^();

METHOD PROTECTED OnObjectStateChanged
SUPER^.OnObjectStateChanged();

SyncProperty(E_BACnetPropIdentifier.PropPresentValue, SIZEOF(aPresentValue), ADR(aPresentValue), E_BA_SyncModeRM.eRead);
END_METHOD

METHOD FB_init : BOOL
VAR_INPUT
	bInitRetains : BOOL; // if TRUE, the retain variables are initialized (warm start / cold start)
	bInCopyCode : BOOL;  // if TRUE, the instance afterwards gets moved into the copy code (online change)
END_VAR
eObjectType := E_BACnetObjType.ObjOctetStringValue;
END_METHOD

END_FUNCTION_BLOCK

// POUs/Remote/Objects/Primitive/FB_BACnetRM_Date
{attribute 'enable_dynamic_creation'}
FUNCTION_BLOCK FB_BACnetRM_Date EXTENDS FB_BACnetRM_Object
VAR_OUTPUT
	stPresentValue 	: ST_BA_Date;
END_VAR

SUPER^();

METHOD PROTECTED OnObjectStateChanged
SUPER^.OnObjectStateChanged();

SyncProperty(E_BACnetPropIdentifier.PropPresentValue, SIZEOF(stPresentValue), ADR(stPresentValue), E_BA_SyncModeRM.eRead);
END_METHOD

METHOD FB_init : BOOL
VAR_INPUT
	bInitRetains : BOOL; // if TRUE, the retain variables are initialized (warm start / cold start)
	bInCopyCode : BOOL;  // if TRUE, the instance afterwards gets moved into the copy code (online change)
END_VAR
eObjectType := E_BACnetObjType.ObjDateValue;
END_METHOD

END_FUNCTION_BLOCK

// POUs/Remote/Objects/Primitive/FB_BACnetRM_DateP
{attribute 'enable_dynamic_creation'}
FUNCTION_BLOCK FB_BACnetRM_DateP EXTENDS FB_BACnetRM_Object
VAR_OUTPUT
	stPresentValue 	: ST_BA_Date;
END_VAR

SUPER^();

METHOD PROTECTED OnObjectStateChanged
SUPER^.OnObjectStateChanged();

SyncProperty(E_BACnetPropIdentifier.PropPresentValue, SIZEOF(stPresentValue), ADR(stPresentValue), E_BA_SyncModeRM.eRead);
END_METHOD

METHOD FB_init : BOOL
VAR_INPUT
	bInitRetains : BOOL; // if TRUE, the retain variables are initialized (warm start / cold start)
	bInCopyCode : BOOL;  // if TRUE, the instance afterwards gets moved into the copy code (online change)
END_VAR
eObjectType := E_BACnetObjType.ObjDatePatternValue;
END_METHOD

END_FUNCTION_BLOCK

// POUs/Remote/Objects/Primitive/FB_BACnetRM_DateTime
{attribute 'enable_dynamic_creation'}
FUNCTION_BLOCK FB_BACnetRM_DateTime EXTENDS FB_BACnetRM_Object
VAR_OUTPUT
	stPresentValue 	: ST_BA_DateTime;
END_VAR

SUPER^();

METHOD PROTECTED OnObjectStateChanged
SUPER^.OnObjectStateChanged();

SyncProperty(E_BACnetPropIdentifier.PropPresentValue, SIZEOF(stPresentValue), ADR(stPresentValue), E_BA_SyncModeRM.eRead);
END_METHOD

METHOD FB_init : BOOL
VAR_INPUT
	bInitRetains : BOOL; // if TRUE, the retain variables are initialized (warm start / cold start)
	bInCopyCode : BOOL;  // if TRUE, the instance afterwards gets moved into the copy code (online change)
END_VAR
eObjectType := E_BACnetObjType.ObjDateTimeValue;
END_METHOD

END_FUNCTION_BLOCK

// POUs/Remote/Objects/Primitive/FB_BACnetRM_DateTimeP
{attribute 'enable_dynamic_creation'}
FUNCTION_BLOCK FB_BACnetRM_DateTimeP EXTENDS FB_BACnetRM_Object
VAR_OUTPUT
	stPresentValue 	: ST_BA_DateTime;
END_VAR

SUPER^();

METHOD PROTECTED OnObjectStateChanged
SUPER^.OnObjectStateChanged();

SyncProperty(E_BACnetPropIdentifier.PropPresentValue, SIZEOF(stPresentValue), ADR(stPresentValue), E_BA_SyncModeRM.eRead);
END_METHOD

METHOD FB_init : BOOL
VAR_INPUT
	bInitRetains : BOOL; // if TRUE, the retain variables are initialized (warm start / cold start)
	bInCopyCode : BOOL;  // if TRUE, the instance afterwards gets moved into the copy code (online change)
END_VAR
eObjectType := E_BACnetObjType.ObjDateTimePatternValue;
END_METHOD

END_FUNCTION_BLOCK

// POUs/Remote/Objects/Primitive/FB_BACnetRM_Int
{attribute 'enable_dynamic_creation'}
FUNCTION_BLOCK FB_BACnetRM_Int EXTENDS FB_BACnetRM_Object
VAR_OUTPUT
	nPresentValue 	: DINT;
END_VAR

SUPER^();

METHOD PROTECTED OnObjectStateChanged
SUPER^.OnObjectStateChanged();

SyncProperty(E_BACnetPropIdentifier.PropPresentValue, SIZEOF(nPresentValue), ADR(nPresentValue), E_BA_SyncModeRM.eRead);
END_METHOD

METHOD FB_init : BOOL
VAR_INPUT
	bInitRetains : BOOL; // if TRUE, the retain variables are initialized (warm start / cold start)
	bInCopyCode : BOOL;  // if TRUE, the instance afterwards gets moved into the copy code (online change)
END_VAR
eObjectType := E_BACnetObjType.ObjIntegerValue;
END_METHOD

END_FUNCTION_BLOCK

// POUs/Remote/Objects/Primitive/FB_BACnetRM_LAV
{attribute 'enable_dynamic_creation'}
FUNCTION_BLOCK FB_BACnetRM_LAV EXTENDS FB_BACnetRM_Object
VAR_OUTPUT
	fPresentValue 	: LREAL;
END_VAR

SUPER^();

METHOD PROTECTED OnObjectStateChanged
SUPER^.OnObjectStateChanged();

SyncProperty(E_BACnetPropIdentifier.PropPresentValue, SIZEOF(fPresentValue), ADR(fPresentValue), E_BA_SyncModeRM.eRead);
END_METHOD

METHOD FB_init : BOOL
VAR_INPUT
	bInitRetains : BOOL; // if TRUE, the retain variables are initialized (warm start / cold start)
	bInCopyCode : BOOL;  // if TRUE, the instance afterwards gets moved into the copy code (online change)
END_VAR
eObjectType := E_BACnetObjType.ObjLargeAnalogValue;
END_METHOD

END_FUNCTION_BLOCK

// POUs/Remote/Objects/Primitive/FB_BACnetRM_String
{attribute 'enable_dynamic_creation'}
FUNCTION_BLOCK FB_BACnetRM_String EXTENDS FB_BACnetRM_Object
VAR_OUTPUT
	sPresentValue 	: STRING;
END_VAR

SUPER^();

METHOD PROTECTED OnObjectStateChanged
SUPER^.OnObjectStateChanged();

SyncProperty(E_BACnetPropIdentifier.PropPresentValue, SIZEOF(sPresentValue), ADR(sPresentValue), E_BA_SyncModeRM.eRead);
END_METHOD

METHOD FB_init : BOOL
VAR_INPUT
	bInitRetains : BOOL; // if TRUE, the retain variables are initialized (warm start / cold start)
	bInCopyCode : BOOL;  // if TRUE, the instance afterwards gets moved into the copy code (online change)
END_VAR
eObjectType := E_BACnetObjType.ObjCharacterStringValue;
END_METHOD

END_FUNCTION_BLOCK

// POUs/Remote/Objects/Primitive/FB_BACnetRM_Time
{attribute 'enable_dynamic_creation'}
FUNCTION_BLOCK FB_BACnetRM_Time EXTENDS FB_BACnetRM_Object
VAR_OUTPUT
	stPresentValue 	: ST_BA_Time;
END_VAR

SUPER^();

METHOD PROTECTED OnObjectStateChanged
SUPER^.OnObjectStateChanged();

SyncProperty(E_BACnetPropIdentifier.PropPresentValue, SIZEOF(stPresentValue), ADR(stPresentValue), E_BA_SyncModeRM.eRead);
END_METHOD

METHOD FB_init : BOOL
VAR_INPUT
	bInitRetains : BOOL; // if TRUE, the retain variables are initialized (warm start / cold start)
	bInCopyCode : BOOL;  // if TRUE, the instance afterwards gets moved into the copy code (online change)
END_VAR
eObjectType := E_BACnetObjType.ObjTimeValue;
END_METHOD

END_FUNCTION_BLOCK

// POUs/Remote/Objects/Primitive/FB_BACnetRM_TimeP
{attribute 'enable_dynamic_creation'}
FUNCTION_BLOCK FB_BACnetRM_TimeP EXTENDS FB_BACnetRM_Object
VAR_OUTPUT
	stPresentValue 	: ST_BA_Time;
END_VAR

SUPER^();

METHOD PROTECTED OnObjectStateChanged
SUPER^.OnObjectStateChanged();

SyncProperty(E_BACnetPropIdentifier.PropPresentValue, SIZEOF(stPresentValue), ADR(stPresentValue), E_BA_SyncModeRM.eRead);
END_METHOD

METHOD FB_init : BOOL
VAR_INPUT
	bInitRetains : BOOL; // if TRUE, the retain variables are initialized (warm start / cold start)
	bInCopyCode : BOOL;  // if TRUE, the instance afterwards gets moved into the copy code (online change)
END_VAR
eObjectType := E_BACnetObjType.ObjTimePatternValue;
END_METHOD

END_FUNCTION_BLOCK

// POUs/Remote/Objects/Primitive/FB_BACnetRM_UInt
{attribute 'enable_dynamic_creation'}
FUNCTION_BLOCK FB_BACnetRM_UInt EXTENDS FB_BACnetRM_Object
VAR_OUTPUT
	nPresentValue 	: UDINT;
END_VAR

SUPER^();

METHOD PROTECTED OnObjectStateChanged
SUPER^.OnObjectStateChanged();

SyncProperty(E_BACnetPropIdentifier.PropPresentValue, SIZEOF(nPresentValue), ADR(nPresentValue), E_BA_SyncModeRM.eRead);
END_METHOD

METHOD FB_init : BOOL
VAR_INPUT
	bInitRetains : BOOL; // if TRUE, the retain variables are initialized (warm start / cold start)
	bInCopyCode : BOOL;  // if TRUE, the instance afterwards gets moved into the copy code (online change)
END_VAR
eObjectType := E_BACnetObjType.ObjPositiveIntegerValue;
END_METHOD

END_FUNCTION_BLOCK

// POUs/Remote/Properties/FB_BACnetRM_ReadPropertyEx
FUNCTION_BLOCK FB_BACnetRM_ReadPropertyEx EXTENDS FB_BACnetRM_ReadProperty
VAR_INPUT
	nObjectInstance : UDINT;
	eObjectType		: E_BACnetObjType;
END_VAR
VAR_OUTPUT
END_VAR
VAR
	refObj : FB_BACnetRM_Object;
	bRefObjUsed : BOOL;
END_VAR

IF iObject = 0 THEN
	iObject := refObj;
	bRefObjUsed:=TRUE;
END_IF

IF bRefObjUsed THEN
	refObj.ObjectInstance:=nObjectInstance;
	refObj.ObjectType:=eObjectType;
END_IF

SUPER^();

END_FUNCTION_BLOCK

// POUs/Remote/Properties/FB_BACnetRM_WritePropertyEx
FUNCTION_BLOCK FB_BACnetRM_WritePropertyEx EXTENDS FB_BACnetRM_WriteProperty
VAR_INPUT
	nObjectInstance : UDINT;
	eObjectType		: E_BACnetObjType;
END_VAR
VAR_OUTPUT
END_VAR
VAR
	refObj : FB_BACnetRM_Object;
	bRefObjUsed : BOOL;
END_VAR

IF iObject = 0 THEN
	iObject := refObj;
	bRefObjUsed:=TRUE;
END_IF

IF bRefObjUsed THEN
	refObj.ObjectInstance:=nObjectInstance;
	refObj.ObjectType:=eObjectType;
END_IF

SUPER^();

END_FUNCTION_BLOCK

// POUs/Remote/Requests/[Internal]/FB_BACnetRM_ReqAckAlarm
{attribute 'c++_compatible'}
{attribute 'enable_dynamic_creation'}
{attribute 'hide'}
FUNCTION_BLOCK FB_BACnetRM_ReqAckAlarm EXTENDS FB_BACnetRM_ReqBase IMPLEMENTS ITcIoBACnetServiceResponseSink
VAR_INPUT
	sMsg : STRING;
	eAckEvent : E_BACnet_EventState;
END_VAR
VAR_OUTPUT
	bTsReady : BOOL;
	bReady : BOOL;
END_VAR
VAR
	req : AcknowledgeAlarmRequest;
	readTsReq : FB_BACnetRM_ReqRead;
	eventTs : ST_BACnet_EventTimeStamps;
END_VAR

IF NOT bTsReady THEN
	bTsReady := readTsReq.bReady;
END_IF

{attribute 'c++_compatible'}
{attribute 'minimal_input_size' := '4'}
{attribute 'pack_mode' := '4'}
{attribute 'hide'}
METHOD OnSendPropertyDataRequest : HRESULT
VAR_INPUT
	pResult	: POINTER TO SendDataRequestResult;
END_VAR
IF (pResult <> 0) THEN
	IF F_BACnetRM_IsErrorSet(pResult) THEN
		bReady := FALSE;
		OnSendPropertyDataRequest:=S_FALSE;
	ELSE
		bReady := FALSE;	
	END_IF
END_IF
END_METHOD

{attribute 'hide'}
METHOD Send : BOOL
VAR
	_ClTmp : ITcIoBACnetPlcClient;
END_VAR
IF Valid THEN
	req.acknowledgingProcessIdentifier := 0;
	req.eventObjectIdentifier := iObject.ObjectID;
	req.acknowledgmentSource := sMsg;
	req.eventStateAcknowledged := eAckEvent;
	IF eAckEvent = E_BACnet_EventState.eNormal THEN
		MEMCPY(ADR(req.timeStamp),ADR(eventTs.toNormal), SIZEOF(ST_BACnet_TimeStampDateTime));
	ELSIF eAckEvent = E_BACnet_EventState.eFault THEN
		MEMCPY(ADR(req.timeStamp),ADR(eventTs.toFault), SIZEOF(ST_BACnet_TimeStampDateTime));
	ELSE
		MEMCPY(ADR(req.timeStamp),ADR(eventTs.toOffNormal), SIZEOF(ST_BACnet_TimeStampDateTime));
	END_IF
	
	_ClTmp := Client.iClient;
	
	IF S_OK = _ClTmp.AcknowledgeAlarm(ADR(req), Client.ObjectInstance, THIS^) THEN
		Send:=TRUE;
	END_IF
END_IF
END_METHOD

{attribute 'c++_compatible'}
{attribute 'minimal_input_size' := '4'}
{attribute 'pack_mode' := '4'}
{attribute 'hide'}
METHOD TcAddRef : UDINT
END_METHOD

{attribute 'c++_compatible'}
{attribute 'minimal_input_size' := '4'}
{attribute 'pack_mode' := '4'}
{attribute 'hide'}
METHOD TcQueryInterface : HRESULT
VAR_INPUT
	iid	: REFERENCE TO IID;
	pipItf	: POINTER TO PVOID;
END_VAR
VAR
	ipSink : ITcIoBACnetServiceResponseSink;
	ipUnknown : ITcUnknown;	
END_VAR
IF GuidsEqual(ADR(iid), ADR(TC_GLOBAL_IID_LIST.IID_ITcIoBACnetServiceResponseSink)) THEN
	ipSink := THIS^; // cast to interface pointer
	pipItf^ := ITCUNKNOWN_TO_PVOID(ipSink);
	TcAddRef();
	TcQueryInterface := S_OK;
ELSIF GuidsEqual(ADR(iid), ADR(TC_GLOBAL_IID_LIST.IID_ITcUnknown)) THEN
	ipUnknown := THIS^; // cast to interface pointer
	pipItf^ := ITCUNKNOWN_TO_PVOID(ipUnknown);
	TcAddRef();
	TcQueryInterface := S_OK;
ELSE
	TcQueryInterface := E_HRESULTAdsErr.NOINTERFACE ; //Call super if this fb extends some other
END_IF
END_METHOD

{attribute 'c++_compatible'}
{attribute 'minimal_input_size' := '4'}
{attribute 'pack_mode' := '4'}
{attribute 'hide'}
METHOD TcRelease : UDINT
END_METHOD

METHOD PRIVATE UpdateTimeStamp : BOOL
VAR_INPUT
END_VAR
IF Valid THEN
	readTsReq(Client := Client, iObject:=iObject, ePropID:=E_BACnetPropIdentifier.PropEventTimeStamps, pData:=ADR(eventTs), nData:=SIZEOF(eventTs));
	readTsReq.Send();
ELSE
	// (BETA) ... Output Error
END_IF
END_METHOD

METHOD GetRequestType : E_BACnetRM_RequestType
VAR_INPUT
END_VAR
GetRequestType := E_BACnetRM_RequestType.eAcknowledge;
END_METHOD

METHOD IsReady : BOOL
VAR_INPUT
END_VAR
IsReady := bReady;
END_METHOD

END_FUNCTION_BLOCK

// POUs/Remote/Requests/[Internal]/FB_BACnetRM_ReqListAdd
{attribute 'c++_compatible'}
{attribute 'enable_dynamic_creation'}
{attribute 'hide'}
FUNCTION_BLOCK FB_BACnetRM_ReqListAdd EXTENDS FB_BACnetRM_ReqBasic
VAR_INPUT
	ePropID : E_BACnetPropIdentifier;
	pData : PVOID;
	nData : UDINT;
END_VAR
VAR 
	req : SendDataRequest;
END_VAR

IF NOT __ISVALIDREF(Client) THEN
	bError:=TRUE;
END_IF

SUPER^();

{attribute 'hide'}
METHOD Send : BOOL
IF Valid THEN
	IF stReq = 0 THEN
		req.service := E_BACnetConfirmedService.SrvAddListElement;
		req.objectIdentifier := iObject.ObjectID;
		req.propertyIdentifier := ePropID;
		req.pData := pData;
		req.nData := nData;
		req.deviceId := Client.ObjectInstance;
		stReq := ADR(req);
	END_IF
	
	Send:=SUPER^.Send();
END_IF
END_METHOD

METHOD PROTECTED ProcessResult : HRESULT
VAR_INPUT
	pResult	: POINTER TO SendDataRequestResult;
END_VAR
bReady:=TRUE;
ProcessResult:=S_OK;
END_METHOD

METHOD GetRequestType : E_BACnetRM_RequestType
VAR_INPUT
END_VAR
GetRequestType := E_BACnetRM_RequestType.eAddListElement;
END_METHOD

METHOD IsReady : BOOL
VAR_INPUT
END_VAR
IsReady := bReady;
END_METHOD

END_FUNCTION_BLOCK

// POUs/Remote/Requests/[Internal]/FB_BACnetRM_ReqListRem
{attribute 'c++_compatible'}
{attribute 'enable_dynamic_creation'}
{attribute 'hide'}
FUNCTION_BLOCK FB_BACnetRM_ReqListRem EXTENDS FB_BACnetRM_ReqBasic
VAR_INPUT
	ePropID : E_BACnetPropIdentifier;
	pData : PVOID;
	nData : UDINT;
END_VAR
VAR 
	req : SendDataRequest;
END_VAR

IF NOT __ISVALIDREF(Client) THEN
	bError:=TRUE;
END_IF

SUPER^();

{attribute 'hide'}
METHOD Send : BOOL
IF Valid THEN
	IF stReq = 0 THEN
		req.service := E_BACnetConfirmedService.SrvRemoveListElement;
		req.objectIdentifier := iObject.ObjectID;
		req.propertyIdentifier := ePropID;
		req.pData := pData;
		req.nData := nData;
		req.deviceId := Client.ObjectInstance;
		stReq := ADR(req);
	END_IF
	
	Send:=SUPER^.Send();
END_IF
END_METHOD

METHOD PROTECTED ProcessResult : HRESULT
VAR_INPUT
	pResult	: POINTER TO SendDataRequestResult;
END_VAR
bReady:=TRUE;
ProcessResult:=S_OK;
END_METHOD

METHOD GetRequestType : E_BACnetRM_RequestType
VAR_INPUT
END_VAR
GetRequestType := E_BACnetRM_RequestType.eRemoveListElement;
END_METHOD

END_FUNCTION_BLOCK
